LIN {X -0.058,Y -138.324,Z 1253.054,A 0.000,B 0.000,C 90.000,E1 189.670} C_DIS
LIN {X -0.054,Y -139.455,Z 1253.007,A 0.000,B 0.000,C 90.000,E1 181.260} C_DIS
LIN {X 0.026,Y -141.003,Z 1252.976,A 0.000,B 0.000,C 90.000,E1 175.641} C_DIS
LIN {X -0.024,Y -142.757,Z 1252.955,A 0.000,B 0.000,C 90.000,E1 171.951} C_DIS
LIN {X -0.068,Y -145.160,Z 1252.930,A 0.000,B 0.000,C 90.000,E1 167.353} C_DIS
LIN {X -0.076,Y -147.782,Z 1252.909,A 0.000,B 0.000,C 90.000,E1 163.685} C_DIS
LIN {X 0.003,Y -150.461,Z 1252.889,A 0.000,B 0.000,C 90.000,E1 160.007} C_DIS
LIN {X 0.078,Y -153.912,Z 1252.869,A 0.000,B 0.000,C 90.000,E1 156.357} C_DIS
LIN {X 0.002,Y -157.323,Z 1252.849,A 0.000,B 0.000,C 90.000,E1 152.794} C_DIS
LIN {X 0.086,Y -161.512,Z 1252.829,A 0.000,B 0.000,C 90.000,E1 149.203} C_DIS
LIN {X -0.037,Y -165.711,Z 1252.809,A 0.000,B 0.000,C 90.000,E1 145.722} C_DIS
LIN {X 0.088,Y -170.657,Z 1252.790,A 0.000,B 0.000,C 90.000,E1 142.190} C_DIS
LIN {X 0.001,Y -175.532,Z 1252.771,A 0.000,B 0.000,C 90.000,E1 138.771} C_DIS
LIN {X -0.005,Y -181.152,Z 1252.752,A 0.000,B 0.000,C 90.000,E1 135.364} C_DIS
LIN {X -0.007,Y -186.606,Z 1252.733,A 0.000,B 0.000,C 90.000,E1 132.000} C_DIS
LIN {X 0.063,Y -191.215,Z 1252.719,A 0.000,B 0.000,C 90.000,E1 129.483} C_DIS
LIN {X -0.014,Y -197.028,Z 1252.701,A 0.000,B 0.000,C 90.000,E1 126.217} C_DIS
LIN {X 0.090,Y -200.353,Z 1252.692,A 0.000,B 0.000,C 90.000,E1 124.532} C_DIS
LIN {X 0.088,Y -310.121,Z 1252.692,A 0.000,B 0.000,C 90.000,E1 124.532} C_DIS
LIN {X -0.070,Y -311.835,Z 1252.692,A 0.000,B 0.000,C 90.000,E1 124.532} C_DIS
LIN {X 0.041,Y -316.000,Z 1252.691,A 0.000,B 0.000,C 90.000,E1 124.326} C_DIS
LIN {X 0.153,Y -318.367,Z 1252.690,A 0.000,B 0.000,C 90.000,E1 124.119} C_DIS
LIN {X -0.062,Y -321.599,Z 1252.688,A 0.000,B 0.000,C 90.000,E1 123.785} C_DIS
LIN {X 0.072,Y -323.525,Z 1252.686,A 0.000,B 0.000,C 90.000,E1 123.452} C_DIS
LIN {X -0.064,Y -325.025,Z 1252.684,A 0.000,B 0.000,C 90.000,E1 123.166} C_DIS
LIN {X -0.150,Y -339.403,Z 1252.663,A 0.000,B 0.000,C 90.000,E1 119.411} C_DIS
LIN {X 0.030,Y -351.700,Z 1252.648,A 0.000,B 0.000,C 90.000,E1 116.616} C_DIS
LIN {X 0.098,Y -365.488,Z 1252.633,A 0.000,B 0.000,C 90.000,E1 113.898} C_DIS
LIN {X 0.158,Y -379.088,Z 1252.620,A 0.000,B 0.000,C 90.000,E1 111.535} C_DIS
LIN {X -0.083,Y -394.054,Z 1252.607,A 0.000,B 0.000,C 90.000,E1 109.268} C_DIS
LIN {X 0.163,Y -410.491,Z 1252.594,A 0.000,B 0.000,C 90.000,E1 106.985} C_DIS
LIN {X -0.097,Y -428.516,Z 1252.582,A 0.000,B 0.000,C 90.000,E1 104.828} C_DIS
LIN {X -0.031,Y -448.086,Z 1252.571,A 0.000,B 0.000,C 90.000,E1 102.703} C_DIS
LIN {X 0.153,Y -468.363,Z 1252.560,A 0.000,B 0.000,C 90.000,E1 100.725} C_DIS
LIN {X 0.224,Y -473.517,Z 1252.557,A 0.000,B 0.000,C 90.000,E1 100.254} C_DIS
LIN {X -0.170,Y -475.724,Z 1252.556,A 0.000,B 0.000,C 90.000,E1 100.074} C_DIS
LIN {X -0.179,Y -477.397,Z 1252.555,A 0.000,B 0.000,C 90.000,E1 99.849} C_DIS
LIN {X 0.161,Y -478.807,Z 1252.553,A 0.000,B 0.000,C 90.000,E1 99.557} C_DIS
LIN {X 0.031,Y -479.855,Z 1252.552,A 0.000,B 0.000,C 90.000,E1 99.321} C_DIS
LIN {X 0.182,Y -481.069,Z 1252.549,A 0.000,B 0.000,C 90.000,E1 98.803} C_DIS
LIN {X -0.135,Y -481.271,Z 1252.546,A 0.000,B 0.000,C 90.000,E1 98.341} C_DIS
LIN {X 0.100,Y -480.495,Z 1252.543,A 0.000,B 0.000,C 90.000,E1 97.814} C_DIS
LIN {X -0.207,Y -478.616,Z 1252.541,A 0.000,B 0.000,C 90.000,E1 97.352} C_DIS
LIN {X 0.083,Y -477.147,Z 1252.539,A 0.000,B 0.000,C 90.000,E1 97.068} C_DIS
LIN {X 0.209,Y -455.290,Z 1252.522,A 0.000,B 0.000,C 90.000,E1 94.012} C_DIS
LIN {X -0.077,Y -434.881,Z 1252.505,A 0.000,B 0.000,C 90.000,E1 90.917} C_DIS
LIN {X -0.165,Y -416.705,Z 1252.487,A 0.000,B 0.000,C 90.000,E1 87.707} C_DIS
LIN {X 0.075,Y -406.737,Z 1252.476,A 0.000,B 0.000,C 90.000,E1 85.755} C_DIS
LIN {X 0.052,Y -398.078,Z 1252.467,A 0.000,B 0.000,C 90.000,E1 84.090} C_DIS
LIN {X -0.043,Y -387.828,Z 1252.456,A 0.000,B 0.000,C 90.000,E1 82.129} C_DIS
LIN {X 0.121,Y -378.888,Z 1252.447,A 0.000,B 0.000,C 90.000,E1 80.387} C_DIS
LIN {X 0.190,Y -369.652,Z 1252.437,A 0.000,B 0.000,C 90.000,E1 78.634} C_DIS
LIN {X 0.091,Y -360.056,Z 1252.427,A 0.000,B 0.000,C 90.000,E1 76.881} C_DIS
LIN {X -0.076,Y -348.672,Z 1252.416,A 0.000,B 0.000,C 90.000,E1 74.810} C_DIS
LIN {X -0.061,Y -337.274,Z 1252.404,A 0.000,B 0.000,C 90.000,E1 72.670} C_DIS
LIN {X -0.163,Y -323.043,Z 1252.388,A 0.000,B 0.000,C 90.000,E1 69.880} C_DIS
LIN {X 0.099,Y -306.698,Z 1252.368,A 0.000,B 0.000,C 90.000,E1 66.305} C_DIS
LIN {X 0.157,Y -293.245,Z 1252.350,A 0.000,B 0.000,C 90.000,E1 62.999} C_DIS
LIN {X -0.037,Y -281.119,Z 1252.331,A 0.000,B 0.000,C 90.000,E1 59.665} C_DIS
LIN {X 0.048,Y -271.095,Z 1252.314,A 0.000,B 0.000,C 90.000,E1 56.548} C_DIS
LIN {X 0.018,Y -260.896,Z 1252.295,A 0.000,B 0.000,C 90.000,E1 53.050} C_DIS
LIN {X 0.087,Y -251.610,Z 1252.275,A 0.000,B 0.000,C 90.000,E1 49.461} C_DIS
LIN {X 0.138,Y -242.914,Z 1252.255,A 0.000,B 0.000,C 90.000,E1 45.810} C_DIS
LIN {X -0.030,Y -236.363,Z 1252.238,A 0.000,B 0.000,C 90.000,E1 42.894} C_DIS
LIN {X 0.080,Y -228.433,Z 1252.217,A 0.000,B 0.000,C 90.000,E1 39.116} C_DIS
LIN {X 0.051,Y -221.113,Z 1252.196,A 0.000,B 0.000,C 90.000,E1 35.311} C_DIS
LIN {X -0.037,Y -214.422,Z 1252.175,A 0.000,B 0.000,C 90.000,E1 31.465} C_DIS
LIN {X 0.068,Y -208.556,Z 1252.153,A 0.000,B 0.000,C 90.000,E1 27.513} C_DIS
LIN {X -0.025,Y -203.615,Z 1252.131,A 0.000,B 0.000,C 90.000,E1 23.567} C_DIS
LIN {X -0.104,Y -199.415,Z 1252.109,A 0.000,B 0.000,C 90.000,E1 19.577} C_DIS
LIN {X 0.077,Y -195.382,Z 1252.082,A 0.000,B 0.000,C 90.000,E1 14.662} C_DIS
LIN {X -0.039,Y -192.250,Z 1252.050,A 0.000,B 0.000,C 90.000,E1 8.973} C_DIS
LIN {X -0.086,Y -193.147,Z 1251.965,A 0.000,B 0.000,C 90.000,E1 353.799} C_DIS
LIN {X -0.012,Y -196.611,Z 1251.934,A 0.000,B 0.000,C 90.000,E1 348.049} C_DIS
LIN {X -0.074,Y -200.794,Z 1251.906,A 0.000,B 0.000,C 90.000,E1 343.196} C_DIS
LIN {X -0.013,Y -205.052,Z 1251.884,A 0.000,B 0.000,C 90.000,E1 339.156} C_DIS
LIN {X -0.035,Y -210.056,Z 1251.862,A 0.000,B 0.000,C 90.000,E1 335.177} C_DIS
LIN {X -0.114,Y -215.658,Z 1251.840,A 0.000,B 0.000,C 90.000,E1 331.257} C_DIS
LIN {X 0.028,Y -222.004,Z 1251.818,A 0.000,B 0.000,C 90.000,E1 327.327} C_DIS
LIN {X -0.011,Y -228.987,Z 1251.797,A 0.000,B 0.000,C 90.000,E1 323.497} C_DIS
LIN {X 0.032,Y -236.807,Z 1251.776,A 0.000,B 0.000,C 90.000,E1 319.703} C_DIS
LIN {X 0.071,Y -245.561,Z 1251.755,A 0.000,B 0.000,C 90.000,E1 315.972} C_DIS
LIN {X 0.038,Y -254.501,Z 1251.737,A 0.000,B 0.000,C 90.000,E1 312.690} C_DIS
LIN {X 0.007,Y -261.337,Z 1251.725,A 0.000,B 0.000,C 90.000,E1 310.539} C_DIS
LIN {X 0.137,Y -269.058,Z 1251.713,A 0.000,B 0.000,C 90.000,E1 308.382} C_DIS
LIN {X -0.011,Y -276.269,Z 1251.704,A 0.000,B 0.000,C 90.000,E1 306.664} C_DIS
LIN {X 0.035,Y -287.524,Z 1251.690,A 0.000,B 0.000,C 90.000,E1 304.246} C_DIS
LIN {X 0.086,Y -298.162,Z 1251.679,A 0.000,B 0.000,C 90.000,E1 302.212} C_DIS
LIN {X -0.104,Y -308.042,Z 1251.670,A 0.000,B 0.000,C 90.000,E1 300.590} C_DIS
LIN {X -0.090,Y -316.893,Z 1251.663,A 0.000,B 0.000,C 90.000,E1 299.283} C_DIS
LIN {X 0.040,Y -333.695,Z 1251.650,A 0.000,B 0.000,C 90.000,E1 297.052} C_DIS
LIN {X 0.051,Y -354.472,Z 1251.637,A 0.000,B 0.000,C 90.000,E1 294.591} C_DIS
LIN {X 0.129,Y -370.142,Z 1251.627,A 0.000,B 0.000,C 90.000,E1 292.823} C_DIS
LIN {X 0.044,Y -382.927,Z 1251.619,A 0.000,B 0.000,C 90.000,E1 291.408} C_DIS
LIN {X -0.151,Y -400.960,Z 1251.608,A 0.000,B 0.000,C 90.000,E1 289.450} C_DIS
LIN {X 0.050,Y -416.174,Z 1251.599,A 0.000,B 0.000,C 90.000,E1 287.819} C_DIS
LIN {X 0.207,Y -425.892,Z 1251.593,A 0.000,B 0.000,C 90.000,E1 286.732} C_DIS
LIN {X -0.128,Y -432.798,Z 1251.589,A 0.000,B 0.000,C 90.000,E1 285.969} C_DIS
LIN {X 0.122,Y -439.139,Z 1251.584,A 0.000,B 0.000,C 90.000,E1 285.134} C_DIS
LIN {X -0.002,Y -444.874,Z 1251.580,A 0.000,B 0.000,C 90.000,E1 284.356} C_DIS
LIN {X -0.185,Y -449.960,Z 1251.575,A 0.000,B 0.000,C 90.000,E1 283.592} C_DIS
LIN {X 0.114,Y -454.343,Z 1251.571,A 0.000,B 0.000,C 90.000,E1 282.771} C_DIS
LIN {X 0.017,Y -458.046,Z 1251.567,A 0.000,B 0.000,C 90.000,E1 282.007} C_DIS
LIN {X -0.055,Y -461.090,Z 1251.562,A 0.000,B 0.000,C 90.000,E1 281.243} C_DIS
LIN {X 0.056,Y -462.821,Z 1251.560,A 0.000,B 0.000,C 90.000,E1 280.715} C_DIS
LIN {X 0.095,Y -464.245,Z 1251.557,A 0.000,B 0.000,C 90.000,E1 280.197} C_DIS
LIN {X 0.228,Y -465.421,Z 1251.554,A 0.000,B 0.000,C 90.000,E1 279.670} C_DIS
LIN {X -0.170,Y -466.301,Z 1251.551,A 0.000,B 0.000,C 90.000,E1 279.208} C_DIS
LIN {X -0.027,Y -466.922,Z 1251.548,A 0.000,B 0.000,C 90.000,E1 278.681} C_DIS
LIN {X 0.050,Y -467.186,Z 1251.545,A 0.000,B 0.000,C 90.000,E1 278.163} C_DIS
LIN {X 0.133,Y -467.079,Z 1251.543,A 0.000,B 0.000,C 90.000,E1 277.644} C_DIS
LIN {X 0.218,Y -466.525,Z 1251.540,A 0.000,B 0.000,C 90.000,E1 277.125} C_DIS
LIN {X -0.159,Y -465.542,Z 1251.537,A 0.000,B 0.000,C 90.000,E1 276.663} C_DIS
LIN {X -0.076,Y -464.136,Z 1251.534,A 0.000,B 0.000,C 90.000,E1 276.144} C_DIS
LIN {X -0.174,Y -461.221,Z 1251.530,A 0.000,B 0.000,C 90.000,E1 275.391} C_DIS
LIN {X -0.156,Y -458.859,Z 1251.527,A 0.000,B 0.000,C 90.000,E1 274.878} C_DIS
LIN {X -0.114,Y -455.967,Z 1251.524,A 0.000,B 0.000,C 90.000,E1 274.359} C_DIS
LIN {X -0.088,Y -452.395,Z 1251.521,A 0.000,B 0.000,C 90.000,E1 273.841} C_DIS
LIN {X -0.110,Y -447.800,Z 1251.518,A 0.000,B 0.000,C 90.000,E1 273.326} C_DIS
LIN {X 0.121,Y -445.050,Z 1251.517,A 0.000,B 0.000,C 90.000,E1 273.037} C_DIS
LIN {X -0.100,Y -438.896,Z 1251.514,A 0.000,B 0.000,C 90.000,E1 272.579} C_DIS
LIN {X -0.209,Y -432.234,Z 1251.512,A 0.000,B 0.000,C 90.000,E1 272.178} C_DIS
LIN {X -0.199,Y -425.256,Z 1251.510,A 0.000,B 0.000,C 90.000,E1 271.833} C_DIS
LIN {X -0.191,Y -418.174,Z 1251.508,A 0.000,B 0.000,C 90.000,E1 271.547} C_DIS
LIN {X -0.160,Y -407.620,Z 1251.507,A 0.000,B 0.000,C 90.000,E1 271.203} C_DIS
LIN {X 0.154,Y -400.372,Z 1251.505,A 0.000,B 0.000,C 90.000,E1 270.974} C_DIS
LIN {X -0.113,Y -393.101,Z 1251.505,A 0.000,B 0.000,C 90.000,E1 270.859} C_DIS
LIN {X -0.171,Y -384.846,Z 1251.504,A 0.000,B 0.000,C 90.000,E1 270.745} C_DIS
LIN {X 0.169,Y -372.232,Z 1251.503,A 0.000,B 0.000,C 90.000,E1 270.573} C_DIS
LIN {X -0.023,Y -363.644,Z 1251.503,A 0.000,B 0.000,C 90.000,E1 270.573} C_DIS
LIN {X -0.036,Y -181.556,Z 1251.503,A 0.000,B 0.000,C 90.000,E1 270.573} C_DIS
LIN {X -0.072,Y -181.282,Z 1251.494,A 0.000,B 0.000,C 90.000,E1 268.854} C_DIS
LIN {X -0.023,Y -180.907,Z 1251.475,A 0.000,B 0.000,C 90.000,E1 265.469} C_DIS
LIN {X 0.034,Y -180.733,Z 1251.470,A 0.000,B 0.000,C 90.000,E1 264.609} C_DIS
LIN {X -0.044,Y -178.822,Z 1251.442,A 0.000,B 0.000,C 90.000,E1 259.567} C_DIS
LIN {X 0.037,Y -175.868,Z 1251.414,A 0.000,B 0.000,C 90.000,E1 254.448} C_DIS
LIN {X 0.032,Y -173.837,Z 1251.399,A 0.000,B 0.000,C 90.000,E1 251.891} C_DIS
LIN {X 0.021,Y -171.505,Z 1251.380,A 0.000,B 0.000,C 90.000,E1 248.465} C_DIS
LIN {X 0.007,Y -167.732,Z 1251.356,A 0.000,B 0.000,C 90.000,E1 244.152} C_DIS
LIN {X 0.024,Y -166.429,Z 1251.347,A 0.000,B 0.000,C 90.000,E1 242.410} C_DIS
LIN {X 0.021,Y -163.149,Z 1251.327,A 0.000,B 0.000,C 90.000,E1 238.918} C_DIS
LIN {X -0.013,Y -161.105,Z 1251.313,A 0.000,B 0.000,C 90.000,E1 236.294} C_DIS
LIN {X -0.030,Y -157.831,Z 1251.293,A 0.000,B 0.000,C 90.000,E1 232.763} C_DIS
LIN {X 0.034,Y -155.865,Z 1251.278,A 0.000,B 0.000,C 90.000,E1 230.070} C_DIS
LIN {X 0.089,Y -152.115,Z 1251.253,A 0.000,B 0.000,C 90.000,E1 225.567} C_DIS
LIN {X -0.004,Y -150.365,Z 1251.238,A 0.000,B 0.000,C 90.000,E1 222.894} C_DIS
LIN {X 0.035,Y -147.100,Z 1251.213,A 0.000,B 0.000,C 90.000,E1 218.338} C_DIS
LIN {X 0.029,Y -145.669,Z 1251.198,A 0.000,B 0.000,C 90.000,E1 215.598} C_DIS
LIN {X 0.032,Y -143.051,Z 1251.172,A 0.000,B 0.000,C 90.000,E1 211.003} C_DIS
LIN {X -0.032,Y -141.674,Z 1251.152,A 0.000,B 0.000,C 90.000,E1 207.334} C_DIS
LIN {X 0.077,Y -139.454,Z 1251.116,A 0.000,B 0.000,C 90.000,E1 200.791} C_DIS
LIN {X -0.003,Y -139.188,Z 1251.105,A 0.000,B 0.000,C 90.000,E1 198.960} C_DIS
LIN {X 0.020,Y -138.323,Z 1251.053,A 0.000,B 0.000,C 90.000,E1 189.613} C_DIS
LIN {X 0.028,Y -139.458,Z 1251.007,A 0.000,B 0.000,C 90.000,E1 181.203} C_DIS
LIN {X -0.032,Y -141.012,Z 1250.976,A 0.000,B 0.000,C 90.000,E1 175.641} C_DIS
LIN {X 0.059,Y -142.766,Z 1250.955,A 0.000,B 0.000,C 90.000,E1 171.894} C_DIS
LIN {X 0.014,Y -145.175,Z 1250.929,A 0.000,B 0.000,C 90.000,E1 167.297} C_DIS
LIN {X 0.047,Y -147.797,Z 1250.909,A 0.000,B 0.000,C 90.000,E1 163.614} C_DIS
LIN {X -0.057,Y -150.481,Z 1250.889,A 0.000,B 0.000,C 90.000,E1 160.007} C_DIS
LIN {X 0.016,Y -153.935,Z 1250.869,A 0.000,B 0.000,C 90.000,E1 156.357} C_DIS
LIN {X 0.079,Y -157.346,Z 1250.849,A 0.000,B 0.000,C 90.000,E1 152.743} C_DIS
LIN {X 0.023,Y -161.541,Z 1250.829,A 0.000,B 0.000,C 90.000,E1 149.203} C_DIS
LIN {X 0.036,Y -165.739,Z 1250.809,A 0.000,B 0.000,C 90.000,E1 145.674} C_DIS
LIN {X 0.023,Y -170.692,Z 1250.790,A 0.000,B 0.000,C 90.000,E1 142.190} C_DIS
LIN {X -0.065,Y -175.565,Z 1250.771,A 0.000,B 0.000,C 90.000,E1 138.771} C_DIS
LIN {X 0.054,Y -181.184,Z 1250.752,A 0.000,B 0.000,C 90.000,E1 135.324} C_DIS
LIN {X -0.076,Y -186.643,Z 1250.733,A 0.000,B 0.000,C 90.000,E1 132.000} C_DIS
LIN {X -0.008,Y -191.249,Z 1250.719,A 0.000,B 0.000,C 90.000,E1 129.483} C_DIS
LIN {X 0.073,Y -197.068,Z 1250.701,A 0.000,B 0.000,C 90.000,E1 126.171} C_DIS
LIN {X 0.019,Y -200.395,Z 1250.692,A 0.000,B 0.000,C 90.000,E1 124.532} C_DIS
LIN {X -0.024,Y -309.372,Z 1250.692,A 0.000,B 0.000,C 90.000,E1 124.532} C_DIS
LIN {X 0.075,Y -311.716,Z 1250.692,A 0.000,B 0.000,C 90.000,E1 124.485} C_DIS
LIN {X -0.072,Y -315.998,Z 1250.691,A 0.000,B 0.000,C 90.000,E1 124.326} C_DIS
LIN {X 0.040,Y -318.385,Z 1250.690,A 0.000,B 0.000,C 90.000,E1 124.119} C_DIS
LIN {X -0.178,Y -321.634,Z 1250.688,A 0.000,B 0.000,C 90.000,E1 123.785} C_DIS
LIN {X -0.037,Y -323.561,Z 1250.686,A 0.000,B 0.000,C 90.000,E1 123.452} C_DIS
LIN {X -0.168,Y -325.062,Z 1250.684,A 0.000,B 0.000,C 90.000,E1 123.166} C_DIS
LIN {X 0.039,Y -339.456,Z 1250.663,A 0.000,B 0.000,C 90.000,E1 119.361} C_DIS
LIN {X -0.079,Y -351.762,Z 1250.648,A 0.000,B 0.000,C 90.000,E1 116.616} C_DIS
LIN {X -0.013,Y -365.559,Z 1250.633,A 0.000,B 0.000,C 90.000,E1 113.898} C_DIS
LIN {X 0.045,Y -379.169,Z 1250.620,A 0.000,B 0.000,C 90.000,E1 111.535} C_DIS
LIN {X -0.199,Y -394.145,Z 1250.607,A 0.000,B 0.000,C 90.000,E1 109.268} C_DIS
LIN {X 0.044,Y -410.593,Z 1250.594,A 0.000,B 0.000,C 90.000,E1 106.985} C_DIS
LIN {X 0.196,Y -428.629,Z 1250.582,A 0.000,B 0.000,C 90.000,E1 104.773} C_DIS
LIN {X -0.150,Y -448.207,Z 1250.570,A 0.000,B 0.000,C 90.000,E1 102.703} C_DIS
LIN {X 0.125,Y -468.490,Z 1250.560,A 0.000,B 0.000,C 90.000,E1 100.715} C_DIS
LIN {X 0.109,Y -473.641,Z 1250.557,A 0.000,B 0.000,C 90.000,E1 100.254} C_DIS
LIN {X 0.155,Y -475.811,Z 1250.556,A 0.000,B 0.000,C 90.000,E1 100.018} C_DIS
LIN {X 0.120,Y -477.454,Z 1250.554,A 0.000,B 0.000,C 90.000,E1 99.792} C_DIS
LIN {X -0.010,Y -478.818,Z 1250.553,A 0.000,B 0.000,C 90.000,E1 99.557} C_DIS
LIN {X -0.141,Y -479.829,Z 1250.552,A 0.000,B 0.000,C 90.000,E1 99.321} C_DIS
LIN {X 0.010,Y -480.981,Z 1250.549,A 0.000,B 0.000,C 90.000,E1 98.803} C_DIS
LIN {X 0.239,Y -481.128,Z 1250.546,A 0.000,B 0.000,C 90.000,E1 98.276} C_DIS
LIN {X -0.072,Y -480.294,Z 1250.543,A 0.000,B 0.000,C 90.000,E1 97.814} C_DIS
LIN {X 0.095,Y -478.343,Z 1250.541,A 0.000,B 0.000,C 90.000,E1 97.296} C_DIS
LIN {X -0.090,Y -476.826,Z 1250.539,A 0.000,B 0.000,C 90.000,E1 97.068} C_DIS
LIN {X -0.008,Y -458.494,Z 1250.525,A 0.000,B 0.000,C 90.000,E1 94.531} C_DIS
LIN {X 0.108,Y -439.450,Z 1250.509,A 0.000,B 0.000,C 90.000,E1 91.661} C_DIS
LIN {X -0.094,Y -423.737,Z 1250.495,A 0.000,B 0.000,C 90.000,E1 89.026} C_DIS
LIN {X 0.125,Y -409.273,Z 1250.479,A 0.000,B 0.000,C 90.000,E1 86.274} C_DIS
LIN {X 0.146,Y -400.680,Z 1250.470,A 0.000,B 0.000,C 90.000,E1 84.609} C_DIS
LIN {X 0.102,Y -390.447,Z 1250.459,A 0.000,B 0.000,C 90.000,E1 82.648} C_DIS
LIN {X -0.124,Y -381.591,Z 1250.450,A 0.000,B 0.000,C 90.000,E1 80.971} C_DIS
LIN {X -0.006,Y -372.448,Z 1250.440,A 0.000,B 0.000,C 90.000,E1 79.218} C_DIS
LIN {X -0.026,Y -364.591,Z 1250.432,A 0.000,B 0.000,C 90.000,E1 77.757} C_DIS
LIN {X -0.131,Y -354.893,Z 1250.422,A 0.000,B 0.000,C 90.000,E1 75.992} C_DIS
LIN {X -0.069,Y -343.475,Z 1250.410,A 0.000,B 0.000,C 90.000,E1 73.866} C_DIS
LIN {X -0.089,Y -330.597,Z 1250.397,A 0.000,B 0.000,C 90.000,E1 71.402} C_DIS
LIN {X 0.095,Y -318.159,Z 1250.383,A 0.000,B 0.000,C 90.000,E1 68.847} C_DIS
LIN {X 0.021,Y -302.275,Z 1250.363,A 0.000,B 0.000,C 90.000,E1 65.305} C_DIS
LIN {X 0.061,Y -288.037,Z 1250.343,A 0.000,B 0.000,C 90.000,E1 61.641} C_DIS
LIN {X -0.004,Y -276.307,Z 1250.324,A 0.000,B 0.000,C 90.000,E1 58.250} C_DIS
LIN {X 0.108,Y -266.620,Z 1250.306,A 0.000,B 0.000,C 90.000,E1 55.102} C_DIS
LIN {X -0.121,Y -256.771,Z 1250.287,A 0.000,B 0.000,C 90.000,E1 51.618} C_DIS
LIN {X 0.105,Y -249.482,Z 1250.271,A 0.000,B 0.000,C 90.000,E1 48.690} C_DIS
LIN {X -0.085,Y -240.902,Z 1250.250,A 0.000,B 0.000,C 90.000,E1 45.081} C_DIS
LIN {X 0.049,Y -234.325,Z 1250.234,A 0.000,B 0.000,C 90.000,E1 42.081} C_DIS
LIN {X 0.053,Y -228.007,Z 1250.217,A 0.000,B 0.000,C 90.000,E1 39.072} C_DIS
LIN {X 0.021,Y -220.660,Z 1250.196,A 0.000,B 0.000,C 90.000,E1 35.264} C_DIS
LIN {X 0.041,Y -213.939,Z 1250.174,A 0.000,B 0.000,C 90.000,E1 31.386} C_DIS
LIN {X 0.026,Y -208.073,Z 1250.153,A 0.000,B 0.000,C 90.000,E1 27.462} C_DIS
LIN {X -0.073,Y -203.138,Z 1250.130,A 0.000,B 0.000,C 90.000,E1 23.515} C_DIS
LIN {X 0.093,Y -198.951,Z 1250.108,A 0.000,B 0.000,C 90.000,E1 19.450} C_DIS
LIN {X 0.057,Y -194.943,Z 1250.081,A 0.000,B 0.000,C 90.000,E1 14.592} C_DIS
LIN {X 0.069,Y -191.876,Z 1250.049,A 0.000,B 0.000,C 90.000,E1 8.859} C_DIS
LIN {X 0.094,Y -192.895,Z 1249.965,A 0.000,B 0.000,C 90.000,E1 353.742} C_DIS
LIN {X -0.034,Y -196.381,Z 1249.934,A 0.000,B 0.000,C 90.000,E1 348.049} C_DIS
LIN {X 0.086,Y -200.590,Z 1249.906,A 0.000,B 0.000,C 90.000,E1 343.142} C_DIS
LIN {X 0.022,Y -204.905,Z 1249.884,A 0.000,B 0.000,C 90.000,E1 339.135} C_DIS
LIN {X 0.010,Y -209.920,Z 1249.862,A 0.000,B 0.000,C 90.000,E1 335.153} C_DIS
LIN {X 0.131,Y -215.545,Z 1249.840,A 0.000,B 0.000,C 90.000,E1 331.179} C_DIS
LIN {X -0.025,Y -221.928,Z 1249.818,A 0.000,B 0.000,C 90.000,E1 327.327} C_DIS
LIN {X -0.068,Y -228.914,Z 1249.797,A 0.000,B 0.000,C 90.000,E1 323.497} C_DIS
LIN {X -0.030,Y -236.736,Z 1249.776,A 0.000,B 0.000,C 90.000,E1 319.703} C_DIS
LIN {X 0.005,Y -245.497,Z 1249.755,A 0.000,B 0.000,C 90.000,E1 315.972} C_DIS
LIN {X -0.032,Y -254.428,Z 1249.737,A 0.000,B 0.000,C 90.000,E1 312.690} C_DIS
LIN {X -0.067,Y -261.268,Z 1249.725,A 0.000,B 0.000,C 90.000,E1 310.539} C_DIS
LIN {X 0.060,Y -269.017,Z 1249.713,A 0.000,B 0.000,C 90.000,E1 308.382} C_DIS
LIN {X -0.090,Y -276.247,Z 1249.704,A 0.000,B 0.000,C 90.000,E1 306.664} C_DIS
LIN {X -0.049,Y -287.473,Z 1249.690,A 0.000,B 0.000,C 90.000,E1 304.246} C_DIS
LIN {X -0.002,Y -298.107,Z 1249.679,A 0.000,B 0.000,C 90.000,E1 302.212} C_DIS
LIN {X 0.070,Y -307.988,Z 1249.670,A 0.000,B 0.000,C 90.000,E1 300.541} C_DIS
LIN {X -0.174,Y -316.783,Z 1249.662,A 0.000,B 0.000,C 90.000,E1 299.283} C_DIS
LIN {X 0.011,Y -326.243,Z 1249.655,A 0.000,B 0.000,C 90.000,E1 297.975} C_DIS
LIN {X 0.077,Y -349.262,Z 1249.640,A 0.000,B 0.000,C 90.000,E1 295.155} C_DIS
LIN {X -0.076,Y -365.142,Z 1249.630,A 0.000,B 0.000,C 90.000,E1 293.387} C_DIS
LIN {X 0.197,Y -378.202,Z 1249.622,A 0.000,B 0.000,C 90.000,E1 291.897} C_DIS
LIN {X 0.086,Y -391.038,Z 1249.614,A 0.000,B 0.000,C 90.000,E1 290.482} C_DIS
LIN {X 0.002,Y -411.509,Z 1249.602,A 0.000,B 0.000,C 90.000,E1 288.308} C_DIS
LIN {X -0.059,Y -419.120,Z 1249.597,A 0.000,B 0.000,C 90.000,E1 287.511} C_DIS
LIN {X 0.101,Y -426.431,Z 1249.593,A 0.000,B 0.000,C 90.000,E1 286.677} C_DIS
LIN {X -0.127,Y -433.306,Z 1249.588,A 0.000,B 0.000,C 90.000,E1 285.898} C_DIS
LIN {X 0.125,Y -439.607,Z 1249.584,A 0.000,B 0.000,C 90.000,E1 285.064} C_DIS
LIN {X -0.111,Y -445.318,Z 1249.579,A 0.000,B 0.000,C 90.000,E1 284.300} C_DIS
LIN {X 0.149,Y -450.332,Z 1249.575,A 0.000,B 0.000,C 90.000,E1 283.480} C_DIS
LIN {X 0.015,Y -454.677,Z 1249.571,A 0.000,B 0.000,C 90.000,E1 282.715} C_DIS
LIN {X -0.080,Y -458.304,Z 1249.566,A 0.000,B 0.000,C 90.000,E1 281.951} C_DIS
LIN {X -0.149,Y -461.305,Z 1249.562,A 0.000,B 0.000,C 90.000,E1 281.186} C_DIS
LIN {X -0.035,Y -463.003,Z 1249.559,A 0.000,B 0.000,C 90.000,E1 280.658} C_DIS
LIN {X 0.005,Y -464.401,Z 1249.556,A 0.000,B 0.000,C 90.000,E1 280.141} C_DIS
LIN {X 0.139,Y -465.529,Z 1249.553,A 0.000,B 0.000,C 90.000,E1 279.613} C_DIS
LIN {X -0.257,Y -466.390,Z 1249.551,A 0.000,B 0.000,C 90.000,E1 279.151} C_DIS
LIN {X -0.113,Y -467.018,Z 1249.548,A 0.000,B 0.000,C 90.000,E1 278.624} C_DIS
LIN {X -0.035,Y -467.268,Z 1249.545,A 0.000,B 0.000,C 90.000,E1 278.106} C_DIS
LIN {X 0.049,Y -467.126,Z 1249.542,A 0.000,B 0.000,C 90.000,E1 277.587} C_DIS
LIN {X 0.136,Y -466.567,Z 1249.539,A 0.000,B 0.000,C 90.000,E1 277.068} C_DIS
LIN {X -0.241,Y -465.557,Z 1249.536,A 0.000,B 0.000,C 90.000,E1 276.606} C_DIS
LIN {X -0.157,Y -464.106,Z 1249.534,A 0.000,B 0.000,C 90.000,E1 276.087} C_DIS
LIN {X 0.206,Y -461.146,Z 1249.529,A 0.000,B 0.000,C 90.000,E1 275.277} C_DIS
LIN {X 0.037,Y -457.304,Z 1249.525,A 0.000,B 0.000,C 90.000,E1 274.531} C_DIS
LIN {X -0.192,Y -455.789,Z 1249.524,A 0.000,B 0.000,C 90.000,E1 274.302} C_DIS
LIN {X -0.167,Y -452.094,Z 1249.521,A 0.000,B 0.000,C 90.000,E1 273.784} C_DIS
LIN {X -0.189,Y -447.430,Z 1249.518,A 0.000,B 0.000,C 90.000,E1 273.269} C_DIS
LIN {X -0.031,Y -441.682,Z 1249.515,A 0.000,B 0.000,C 90.000,E1 272.751} C_DIS
LIN {X -0.100,Y -438.490,Z 1249.514,A 0.000,B 0.000,C 90.000,E1 272.522} C_DIS
LIN {X -0.199,Y -431.662,Z 1249.512,A 0.000,B 0.000,C 90.000,E1 272.121} C_DIS
LIN {X -0.145,Y -424.631,Z 1249.510,A 0.000,B 0.000,C 90.000,E1 271.776} C_DIS
LIN {X -0.095,Y -417.504,Z 1249.508,A 0.000,B 0.000,C 90.000,E1 271.489} C_DIS
LIN {X 0.005,Y -407.161,Z 1249.506,A 0.000,B 0.000,C 90.000,E1 271.146} C_DIS
LIN {X 0.186,Y -396.224,Z 1249.505,A 0.000,B 0.000,C 90.000,E1 270.859} C_DIS
LIN {X 0.020,Y -388.400,Z 1249.504,A 0.000,B 0.000,C 90.000,E1 270.745} C_DIS
LIN {X 0.052,Y -379.512,Z 1249.504,A 0.000,B 0.000,C 90.000,E1 270.630} C_DIS
LIN {X -0.077,Y -368.342,Z 1249.503,A 0.000,B 0.000,C 90.000,E1 270.573} C_DIS
LIN {X -0.146,Y -363.509,Z 1249.503,A 0.000,B 0.000,C 90.000,E1 270.573} C_DIS
LIN {X 0.089,Y -181.558,Z 1249.503,A 0.000,B 0.000,C 90.000,E1 270.516} C_DIS
LIN {X 0.066,Y -181.279,Z 1249.493,A 0.000,B 0.000,C 90.000,E1 268.797} C_DIS
LIN {X -0.066,Y -180.907,Z 1249.475,A 0.000,B 0.000,C 90.000,E1 265.469} C_DIS
LIN {X -0.010,Y -180.726,Z 1249.470,A 0.000,B 0.000,C 90.000,E1 264.609} C_DIS
LIN {X 0.087,Y -178.815,Z 1249.442,A 0.000,B 0.000,C 90.000,E1 259.511} C_DIS
LIN {X -0.006,Y -175.860,Z 1249.414,A 0.000,B 0.000,C 90.000,E1 254.448} C_DIS
LIN {X 0.043,Y -173.827,Z 1249.399,A 0.000,B 0.000,C 90.000,E1 251.873} C_DIS
LIN {X -0.022,Y -171.493,Z 1249.380,A 0.000,B 0.000,C 90.000,E1 248.465} C_DIS
LIN {X -0.034,Y -167.721,Z 1249.356,A 0.000,B 0.000,C 90.000,E1 244.152} C_DIS
LIN {X -0.018,Y -166.415,Z 1249.347,A 0.000,B 0.000,C 90.000,E1 242.410} C_DIS
LIN {X -0.019,Y -163.137,Z 1249.327,A 0.000,B 0.000,C 90.000,E1 238.918} C_DIS
LIN {X -0.054,Y -161.091,Z 1249.313,A 0.000,B 0.000,C 90.000,E1 236.294} C_DIS
LIN {X -0.070,Y -157.820,Z 1249.293,A 0.000,B 0.000,C 90.000,E1 232.763} C_DIS
LIN {X -0.007,Y -155.854,Z 1249.278,A 0.000,B 0.000,C 90.000,E1 230.070} C_DIS
LIN {X 0.050,Y -152.104,Z 1249.253,A 0.000,B 0.000,C 90.000,E1 225.567} C_DIS
LIN {X 0.068,Y -150.355,Z 1249.238,A 0.000,B 0.000,C 90.000,E1 222.852} C_DIS
LIN {X -0.003,Y -147.091,Z 1249.213,A 0.000,B 0.000,C 90.000,E1 218.338} C_DIS
LIN {X -0.009,Y -145.662,Z 1249.198,A 0.000,B 0.000,C 90.000,E1 215.598} C_DIS
LIN {X -0.005,Y -143.044,Z 1249.172,A 0.000,B 0.000,C 90.000,E1 211.003} C_DIS
LIN {X -0.005,Y -141.668,Z 1249.152,A 0.000,B 0.000,C 90.000,E1 207.308} C_DIS
LIN {X 0.040,Y -139.451,Z 1249.116,A 0.000,B 0.000,C 90.000,E1 200.791} C_DIS
LIN {X -0.040,Y -139.185,Z 1249.105,A 0.000,B 0.000,C 90.000,E1 198.960} C_DIS
LIN {X -0.017,Y -138.321,Z 1249.053,A 0.000,B 0.000,C 90.000,E1 189.613} C_DIS
LIN {X -0.009,Y -139.462,Z 1249.007,A 0.000,B 0.000,C 90.000,E1 181.203} C_DIS
LIN {X -0.070,Y -141.019,Z 1248.976,A 0.000,B 0.000,C 90.000,E1 175.641} C_DIS
LIN {X 0.026,Y -142.382,Z 1248.960,A 0.000,B 0.000,C 90.000,E1 172.818} C_DIS
LIN {X -0.053,Y -144.613,Z 1248.934,A 0.000,B 0.000,C 90.000,E1 168.229} C_DIS
LIN {X 0.009,Y -147.807,Z 1248.909,A 0.000,B 0.000,C 90.000,E1 163.614} C_DIS
LIN {X 0.045,Y -150.494,Z 1248.889,A 0.000,B 0.000,C 90.000,E1 159.953} C_DIS
LIN {X -0.024,Y -153.950,Z 1248.869,A 0.000,B 0.000,C 90.000,E1 156.357} C_DIS
LIN {X 0.039,Y -157.362,Z 1248.849,A 0.000,B 0.000,C 90.000,E1 152.743} C_DIS
LIN {X -0.018,Y -161.560,Z 1248.829,A 0.000,B 0.000,C 90.000,E1 149.203} C_DIS
LIN {X -0.006,Y -165.758,Z 1248.809,A 0.000,B 0.000,C 90.000,E1 145.674} C_DIS
LIN {X -0.020,Y -170.714,Z 1248.790,A 0.000,B 0.000,C 90.000,E1 142.190} C_DIS
LIN {X 0.023,Y -175.587,Z 1248.771,A 0.000,B 0.000,C 90.000,E1 138.728} C_DIS
LIN {X 0.011,Y -181.204,Z 1248.752,A 0.000,B 0.000,C 90.000,E1 135.324} C_DIS
LIN {X 0.004,Y -186.668,Z 1248.733,A 0.000,B 0.000,C 90.000,E1 131.962} C_DIS
LIN {X -0.053,Y -191.270,Z 1248.719,A 0.000,B 0.000,C 90.000,E1 129.483} C_DIS
LIN {X 0.027,Y -197.094,Z 1248.701,A 0.000,B 0.000,C 90.000,E1 126.171} C_DIS
LIN {X 0.069,Y -200.460,Z 1248.692,A 0.000,B 0.000,C 90.000,E1 124.485} C_DIS
LIN {X 0.055,Y -310.542,Z 1248.692,A 0.000,B 0.000,C 90.000,E1 124.485} C_DIS
LIN {X -0.146,Y -315.875,Z 1248.691,A 0.000,B 0.000,C 90.000,E1 124.326} C_DIS
LIN {X -0.034,Y -318.319,Z 1248.690,A 0.000,B 0.000,C 90.000,E1 124.119} C_DIS
LIN {X 0.195,Y -321.613,Z 1248.688,A 0.000,B 0.000,C 90.000,E1 123.706} C_DIS
LIN {X 0.083,Y -323.544,Z 1248.686,A 0.000,B 0.000,C 90.000,E1 123.420} C_DIS
LIN {X -0.208,Y -325.050,Z 1248.684,A 0.000,B 0.000,C 90.000,E1 123.166} C_DIS
LIN {X 0.026,Y -338.181,Z 1248.665,A 0.000,B 0.000,C 90.000,E1 119.667} C_DIS
LIN {X 0.170,Y -350.335,Z 1248.649,A 0.000,B 0.000,C 90.000,E1 116.873} C_DIS
LIN {X -0.123,Y -363.961,Z 1248.634,A 0.000,B 0.000,C 90.000,E1 114.207} C_DIS
LIN {X -0.111,Y -377.411,Z 1248.621,A 0.000,B 0.000,C 90.000,E1 111.844} C_DIS
LIN {X 0.098,Y -392.214,Z 1248.608,A 0.000,B 0.000,C 90.000,E1 109.504} C_DIS
LIN {X -0.091,Y -408.475,Z 1248.596,A 0.000,B 0.000,C 90.000,E1 107.275} C_DIS
LIN {X -0.005,Y -426.310,Z 1248.584,A 0.000,B 0.000,C 90.000,E1 105.064} C_DIS
LIN {X -0.033,Y -445.733,Z 1248.572,A 0.000,B 0.000,C 90.000,E1 102.939} C_DIS
LIN {X 0.080,Y -465.948,Z 1248.561,A 0.000,B 0.000,C 90.000,E1 100.950} C_DIS
LIN {X 0.060,Y -473.671,Z 1248.557,A 0.000,B 0.000,C 90.000,E1 100.254} C_DIS
LIN {X 0.104,Y -475.802,Z 1248.556,A 0.000,B 0.000,C 90.000,E1 100.018} C_DIS
LIN {X 0.065,Y -477.419,Z 1248.554,A 0.000,B 0.000,C 90.000,E1 99.792} C_DIS
LIN {X -0.065,Y -478.760,Z 1248.553,A 0.000,B 0.000,C 90.000,E1 99.557} C_DIS
LIN {X -0.196,Y -479.752,Z 1248.552,A 0.000,B 0.000,C 90.000,E1 99.321} C_DIS
LIN {X -0.046,Y -480.871,Z 1248.549,A 0.000,B 0.000,C 90.000,E1 98.803} C_DIS
LIN {X 0.183,Y -480.989,Z 1248.546,A 0.000,B 0.000,C 90.000,E1 98.276} C_DIS
LIN {X -0.128,Y -480.126,Z 1248.543,A 0.000,B 0.000,C 90.000,E1 97.814} C_DIS
LIN {X 0.038,Y -478.137,Z 1248.541,A 0.000,B 0.000,C 90.000,E1 97.296} C_DIS
LIN {X -0.148,Y -476.595,Z 1248.539,A 0.000,B 0.000,C 90.000,E1 97.068} C_DIS
LIN {X 0.167,Y -456.485,Z 1248.524,A 0.000,B 0.000,C 90.000,E1 94.245} C_DIS
LIN {X -0.051,Y -435.954,Z 1248.506,A 0.000,B 0.000,C 90.000,E1 91.146} C_DIS
LIN {X -0.106,Y -417.583,Z 1248.488,A 0.000,B 0.000,C 90.000,E1 87.936} C_DIS
LIN {X -0.125,Y -404.792,Z 1248.475,A 0.000,B 0.000,C 90.000,E1 85.469} C_DIS
LIN {X -0.113,Y -394.597,Z 1248.464,A 0.000,B 0.000,C 90.000,E1 83.514} C_DIS
LIN {X 0.158,Y -384.336,Z 1248.453,A 0.000,B 0.000,C 90.000,E1 81.489} C_DIS
LIN {X -0.127,Y -376.839,Z 1248.445,A 0.000,B 0.000,C 90.000,E1 80.095} C_DIS
LIN {X -0.088,Y -367.548,Z 1248.435,A 0.000,B 0.000,C 90.000,E1 78.342} C_DIS
LIN {X 0.129,Y -357.965,Z 1248.425,A 0.000,B 0.000,C 90.000,E1 76.533} C_DIS
LIN {X 0.000,Y -346.526,Z 1248.414,A 0.000,B 0.000,C 90.000,E1 74.448} C_DIS
LIN {X -0.040,Y -333.608,Z 1248.400,A 0.000,B 0.000,C 90.000,E1 72.000} C_DIS
LIN {X -0.189,Y -321.047,Z 1248.386,A 0.000,B 0.000,C 90.000,E1 69.518} C_DIS
LIN {X 0.130,Y -304.915,Z 1248.366,A 0.000,B 0.000,C 90.000,E1 65.921} C_DIS
LIN {X 0.128,Y -290.346,Z 1248.346,A 0.000,B 0.000,C 90.000,E1 62.281} C_DIS
LIN {X -0.009,Y -278.376,Z 1248.327,A 0.000,B 0.000,C 90.000,E1 58.918} C_DIS
LIN {X 0.009,Y -268.486,Z 1248.310,A 0.000,B 0.000,C 90.000,E1 55.801} C_DIS
LIN {X 0.046,Y -258.391,Z 1248.290,A 0.000,B 0.000,C 90.000,E1 52.271} C_DIS
LIN {X 0.002,Y -249.189,Z 1248.271,A 0.000,B 0.000,C 90.000,E1 48.690} C_DIS
LIN {X -0.024,Y -240.593,Z 1248.250,A 0.000,B 0.000,C 90.000,E1 45.040} C_DIS
LIN {X -0.065,Y -233.974,Z 1248.234,A 0.000,B 0.000,C 90.000,E1 42.081} C_DIS
LIN {X -0.023,Y -226.085,Z 1248.213,A 0.000,B 0.000,C 90.000,E1 38.302} C_DIS
LIN {X -0.072,Y -218.814,Z 1248.192,A 0.000,B 0.000,C 90.000,E1 34.485} C_DIS
LIN {X -0.045,Y -212.245,Z 1248.170,A 0.000,B 0.000,C 90.000,E1 30.590} C_DIS
LIN {X 0.074,Y -206.579,Z 1248.148,A 0.000,B 0.000,C 90.000,E1 26.616} C_DIS
LIN {X 0.023,Y -201.784,Z 1248.126,A 0.000,B 0.000,C 90.000,E1 22.642} C_DIS
LIN {X -0.033,Y -197.026,Z 1248.099,A 0.000,B 0.000,C 90.000,E1 17.819} C_DIS
LIN {X -0.057,Y -193.505,Z 1248.072,A 0.000,B 0.000,C 90.000,E1 12.939} C_DIS
LIN {X -0.062,Y -190.839,Z 1248.035,A 0.000,B 0.000,C 90.000,E1 6.372} C_DIS
LIN {X -0.067,Y -192.258,Z 1247.970,A 0.000,B 0.000,C 90.000,E1 354.609} C_DIS
LIN {X -0.071,Y -195.559,Z 1247.938,A 0.000,B 0.000,C 90.000,E1 348.870} C_DIS
LIN {X -0.032,Y -199.595,Z 1247.911,A 0.000,B 0.000,C 90.000,E1 343.976} C_DIS
LIN {X -0.003,Y -203.824,Z 1247.889,A 0.000,B 0.000,C 90.000,E1 339.934} C_DIS
LIN {X 0.059,Y -208.733,Z 1247.866,A 0.000,B 0.000,C 90.000,E1 335.921} C_DIS
LIN {X 0.039,Y -214.249,Z 1247.844,A 0.000,B 0.000,C 90.000,E1 331.975} C_DIS
LIN {X 0.028,Y -220.496,Z 1247.823,A 0.000,B 0.000,C 90.000,E1 328.074} C_DIS
LIN {X 0.130,Y -227.375,Z 1247.801,A 0.000,B 0.000,C 90.000,E1 324.196} C_DIS
LIN {X -0.016,Y -234.994,Z 1247.780,A 0.000,B 0.000,C 90.000,E1 320.436} C_DIS
LIN {X -0.020,Y -243.581,Z 1247.759,A 0.000,B 0.000,C 90.000,E1 316.701} C_DIS
LIN {X 0.053,Y -252.276,Z 1247.741,A 0.000,B 0.000,C 90.000,E1 313.380} C_DIS
LIN {X 0.011,Y -259.986,Z 1247.727,A 0.000,B 0.000,C 90.000,E1 310.862} C_DIS
LIN {X -0.089,Y -267.616,Z 1247.715,A 0.000,B 0.000,C 90.000,E1 308.749} C_DIS
LIN {X 0.125,Y -274.703,Z 1247.705,A 0.000,B 0.000,C 90.000,E1 306.950} C_DIS
LIN {X 0.135,Y -285.757,Z 1247.692,A 0.000,B 0.000,C 90.000,E1 304.532} C_DIS
LIN {X -0.092,Y -296.206,Z 1247.681,A 0.000,B 0.000,C 90.000,E1 302.546} C_DIS
LIN {X -0.051,Y -305.815,Z 1247.672,A 0.000,B 0.000,C 90.000,E1 300.875} C_DIS
LIN {X 0.095,Y -314.406,Z 1247.664,A 0.000,B 0.000,C 90.000,E1 299.539} C_DIS
LIN {X -0.066,Y -323.730,Z 1247.657,A 0.000,B 0.000,C 90.000,E1 298.281} C_DIS
LIN {X 0.080,Y -341.339,Z 1247.645,A 0.000,B 0.000,C 90.000,E1 296.052} C_DIS
LIN {X -0.059,Y -359.821,Z 1247.633,A 0.000,B 0.000,C 90.000,E1 293.951} C_DIS
LIN {X 0.053,Y -375.426,Z 1247.623,A 0.000,B 0.000,C 90.000,E1 292.206} C_DIS
LIN {X -0.064,Y -388.339,Z 1247.615,A 0.000,B 0.000,C 90.000,E1 290.791} C_DIS
LIN {X 0.198,Y -408.872,Z 1247.603,A 0.000,B 0.000,C 90.000,E1 288.544} C_DIS
LIN {X -0.091,Y -419.077,Z 1247.597,A 0.000,B 0.000,C 90.000,E1 287.511} C_DIS
LIN {X 0.079,Y -426.407,Z 1247.593,A 0.000,B 0.000,C 90.000,E1 286.677} C_DIS
LIN {X -0.155,Y -433.273,Z 1247.588,A 0.000,B 0.000,C 90.000,E1 285.898} C_DIS
LIN {X 0.096,Y -439.599,Z 1247.584,A 0.000,B 0.000,C 90.000,E1 285.064} C_DIS
LIN {X -0.140,Y -445.298,Z 1247.579,A 0.000,B 0.000,C 90.000,E1 284.300} C_DIS
LIN {X 0.119,Y -450.316,Z 1247.575,A 0.000,B 0.000,C 90.000,E1 283.480} C_DIS
LIN {X -0.017,Y -454.675,Z 1247.571,A 0.000,B 0.000,C 90.000,E1 282.715} C_DIS
LIN {X -0.111,Y -458.305,Z 1247.566,A 0.000,B 0.000,C 90.000,E1 281.951} C_DIS
LIN {X -0.180,Y -461.280,Z 1247.562,A 0.000,B 0.000,C 90.000,E1 281.186} C_DIS
LIN {X -0.067,Y -462.968,Z 1247.559,A 0.000,B 0.000,C 90.000,E1 280.658} C_DIS
LIN {X -0.027,Y -464.396,Z 1247.556,A 0.000,B 0.000,C 90.000,E1 280.141} C_DIS
LIN {X 0.107,Y -465.535,Z 1247.553,A 0.000,B 0.000,C 90.000,E1 279.613} C_DIS
LIN {X 0.172,Y -466.403,Z 1247.551,A 0.000,B 0.000,C 90.000,E1 279.095} C_DIS
LIN {X -0.145,Y -467.026,Z 1247.548,A 0.000,B 0.000,C 90.000,E1 278.624} C_DIS
LIN {X -0.067,Y -467.289,Z 1247.545,A 0.000,B 0.000,C 90.000,E1 278.106} C_DIS
LIN {X 0.017,Y -467.214,Z 1247.542,A 0.000,B 0.000,C 90.000,E1 277.587} C_DIS
LIN {X 0.104,Y -466.666,Z 1247.539,A 0.000,B 0.000,C 90.000,E1 277.068} C_DIS
LIN {X 0.190,Y -465.697,Z 1247.536,A 0.000,B 0.000,C 90.000,E1 276.549} C_DIS
LIN {X -0.187,Y -464.258,Z 1247.534,A 0.000,B 0.000,C 90.000,E1 276.087} C_DIS
LIN {X 0.176,Y -461.344,Z 1247.529,A 0.000,B 0.000,C 90.000,E1 275.277} C_DIS
LIN {X 0.009,Y -457.513,Z 1247.525,A 0.000,B 0.000,C 90.000,E1 274.531} C_DIS
LIN {X 0.041,Y -454.247,Z 1247.522,A 0.000,B 0.000,C 90.000,E1 274.012} C_DIS
LIN {X 0.027,Y -450.139,Z 1247.519,A 0.000,B 0.000,C 90.000,E1 273.498} C_DIS
LIN {X -0.213,Y -447.688,Z 1247.518,A 0.000,B 0.000,C 90.000,E1 273.269} C_DIS
LIN {X -0.056,Y -441.986,Z 1247.515,A 0.000,B 0.000,C 90.000,E1 272.751} C_DIS
LIN {X -0.128,Y -438.778,Z 1247.514,A 0.000,B 0.000,C 90.000,E1 272.522} C_DIS
LIN {X -0.218,Y -432.022,Z 1247.512,A 0.000,B 0.000,C 90.000,E1 272.121} C_DIS
LIN {X -0.162,Y -425.079,Z 1247.510,A 0.000,B 0.000,C 90.000,E1 271.776} C_DIS
LIN {X -0.092,Y -418.140,Z 1247.508,A 0.000,B 0.000,C 90.000,E1 271.489} C_DIS
LIN {X -0.120,Y -411.154,Z 1247.507,A 0.000,B 0.000,C 90.000,E1 271.260} C_DIS
LIN {X -0.098,Y -400.472,Z 1247.505,A 0.000,B 0.000,C 90.000,E1 270.974} C_DIS
LIN {X 0.037,Y -393.009,Z 1247.505,A 0.000,B 0.000,C 90.000,E1 270.802} C_DIS
LIN {X -0.040,Y -384.792,Z 1247.504,A 0.000,B 0.000,C 90.000,E1 270.688} C_DIS
LIN {X 0.049,Y -375.546,Z 1247.503,A 0.000,B 0.000,C 90.000,E1 270.573} C_DIS
LIN {X 0.082,Y -362.162,Z 1247.503,A 0.000,B 0.000,C 90.000,E1 270.516} C_DIS
LIN {X 0.018,Y -181.562,Z 1247.503,A 0.000,B 0.000,C 90.000,E1 270.516} C_DIS
LIN {X -0.006,Y -181.274,Z 1247.493,A 0.000,B 0.000,C 90.000,E1 268.797} C_DIS
LIN {X 0.042,Y -180.906,Z 1247.475,A 0.000,B 0.000,C 90.000,E1 265.412} C_DIS
LIN {X -0.081,Y -180.716,Z 1247.470,A 0.000,B 0.000,C 90.000,E1 264.609} C_DIS
LIN {X 0.016,Y -178.803,Z 1247.442,A 0.000,B 0.000,C 90.000,E1 259.511} C_DIS
LIN {X 0.093,Y -175.848,Z 1247.413,A 0.000,B 0.000,C 90.000,E1 254.393} C_DIS
LIN {X 0.052,Y -172.584,Z 1247.390,A 0.000,B 0.000,C 90.000,E1 250.134} C_DIS
LIN {X 0.068,Y -171.474,Z 1247.380,A 0.000,B 0.000,C 90.000,E1 248.411} C_DIS
LIN {X 0.048,Y -167.704,Z 1247.356,A 0.000,B 0.000,C 90.000,E1 244.101} C_DIS
LIN {X 0.061,Y -166.391,Z 1247.347,A 0.000,B 0.000,C 90.000,E1 242.359} C_DIS
LIN {X 0.052,Y -163.118,Z 1247.327,A 0.000,B 0.000,C 90.000,E1 238.869} C_DIS
LIN {X 0.102,Y -161.067,Z 1247.313,A 0.000,B 0.000,C 90.000,E1 236.215} C_DIS
LIN {X -0.011,Y -157.800,Z 1247.293,A 0.000,B 0.000,C 90.000,E1 232.718} C_DIS
LIN {X -0.072,Y -155.836,Z 1247.278,A 0.000,B 0.000,C 90.000,E1 230.070} C_DIS
LIN {X -0.015,Y -152.086,Z 1247.253,A 0.000,B 0.000,C 90.000,E1 225.567} C_DIS
LIN {X 0.004,Y -150.337,Z 1247.238,A 0.000,B 0.000,C 90.000,E1 222.852} C_DIS
LIN {X 0.024,Y -147.077,Z 1247.213,A 0.000,B 0.000,C 90.000,E1 218.302} C_DIS
LIN {X -0.071,Y -145.650,Z 1247.198,A 0.000,B 0.000,C 90.000,E1 215.598} C_DIS
LIN {X -0.068,Y -143.033,Z 1247.172,A 0.000,B 0.000,C 90.000,E1 211.003} C_DIS
LIN {X 0.059,Y -141.657,Z 1247.152,A 0.000,B 0.000,C 90.000,E1 207.257} C_DIS
LIN {X -0.022,Y -139.447,Z 1247.115,A 0.000,B 0.000,C 90.000,E1 200.791} C_DIS
LIN {X 0.031,Y -139.180,Z 1247.105,A 0.000,B 0.000,C 90.000,E1 198.906} C_DIS
LIN {X 0.059,Y -138.320,Z 1247.053,A 0.000,B 0.000,C 90.000,E1 189.557} C_DIS
LIN {X 0.068,Y -139.465,Z 1247.006,A 0.000,B 0.000,C 90.000,E1 181.146} C_DIS
LIN {X 0.010,Y -141.029,Z 1246.975,A 0.000,B 0.000,C 90.000,E1 175.584} C_DIS
LIN {X -0.036,Y -142.396,Z 1246.960,A 0.000,B 0.000,C 90.000,E1 172.818} C_DIS
LIN {X 0.026,Y -144.628,Z 1246.934,A 0.000,B 0.000,C 90.000,E1 168.173} C_DIS
LIN {X -0.055,Y -147.823,Z 1246.909,A 0.000,B 0.000,C 90.000,E1 163.614} C_DIS
LIN {X 0.031,Y -150.514,Z 1246.889,A 0.000,B 0.000,C 90.000,E1 159.934} C_DIS
LIN {X 0.052,Y -153.976,Z 1246.868,A 0.000,B 0.000,C 90.000,E1 156.305} C_DIS
LIN {X -0.028,Y -157.388,Z 1246.849,A 0.000,B 0.000,C 90.000,E1 152.743} C_DIS
LIN {X -0.086,Y -161.591,Z 1246.829,A 0.000,B 0.000,C 90.000,E1 149.203} C_DIS
LIN {X -0.075,Y -165.789,Z 1246.809,A 0.000,B 0.000,C 90.000,E1 145.674} C_DIS
LIN {X -0.090,Y -170.751,Z 1246.790,A 0.000,B 0.000,C 90.000,E1 142.190} C_DIS
LIN {X 0.068,Y -175.623,Z 1246.771,A 0.000,B 0.000,C 90.000,E1 138.690} C_DIS
LIN {X -0.062,Y -181.238,Z 1246.752,A 0.000,B 0.000,C 90.000,E1 135.324} C_DIS
LIN {X 0.069,Y -186.708,Z 1246.733,A 0.000,B 0.000,C 90.000,E1 131.919} C_DIS
LIN {X 0.020,Y -191.308,Z 1246.719,A 0.000,B 0.000,C 90.000,E1 129.439} C_DIS
LIN {X -0.049,Y -197.137,Z 1246.701,A 0.000,B 0.000,C 90.000,E1 126.171} C_DIS
LIN {X -0.007,Y -200.503,Z 1246.692,A 0.000,B 0.000,C 90.000,E1 124.485} C_DIS
LIN {X -0.064,Y -310.193,Z 1246.692,A 0.000,B 0.000,C 90.000,E1 124.485} C_DIS
LIN {X -0.006,Y -315.878,Z 1246.690,A 0.000,B 0.000,C 90.000,E1 124.278} C_DIS
LIN {X -0.156,Y -318.343,Z 1246.689,A 0.000,B 0.000,C 90.000,E1 124.119} C_DIS
LIN {X 0.072,Y -321.653,Z 1246.687,A 0.000,B 0.000,C 90.000,E1 123.706} C_DIS
LIN {X -0.034,Y -323.584,Z 1246.686,A 0.000,B 0.000,C 90.000,E1 123.420} C_DIS
LIN {X 0.131,Y -325.092,Z 1246.684,A 0.000,B 0.000,C 90.000,E1 123.086} C_DIS
LIN {X -0.088,Y -338.239,Z 1246.665,A 0.000,B 0.000,C 90.000,E1 119.667} C_DIS
LIN {X 0.054,Y -350.402,Z 1246.649,A 0.000,B 0.000,C 90.000,E1 116.873} C_DIS
LIN {X 0.091,Y -364.038,Z 1246.634,A 0.000,B 0.000,C 90.000,E1 114.155} C_DIS
LIN {X -0.232,Y -377.498,Z 1246.621,A 0.000,B 0.000,C 90.000,E1 111.844} C_DIS
LIN {X -0.026,Y -392.312,Z 1246.608,A 0.000,B 0.000,C 90.000,E1 109.504} C_DIS
LIN {X 0.172,Y -408.585,Z 1246.596,A 0.000,B 0.000,C 90.000,E1 107.221} C_DIS
LIN {X -0.135,Y -426.432,Z 1246.584,A 0.000,B 0.000,C 90.000,E1 105.064} C_DIS
LIN {X -0.163,Y -445.866,Z 1246.572,A 0.000,B 0.000,C 90.000,E1 102.939} C_DIS
LIN {X -0.045,Y -466.086,Z 1246.561,A 0.000,B 0.000,C 90.000,E1 100.950} C_DIS
LIN {X -0.064,Y -473.793,Z 1246.557,A 0.000,B 0.000,C 90.000,E1 100.254} C_DIS
LIN {X -0.029,Y -475.867,Z 1246.556,A 0.000,B 0.000,C 90.000,E1 100.018} C_DIS
LIN {X -0.074,Y -477.444,Z 1246.554,A 0.000,B 0.000,C 90.000,E1 99.792} C_DIS
LIN {X -0.205,Y -478.746,Z 1246.553,A 0.000,B 0.000,C 90.000,E1 99.557} C_DIS
LIN {X 0.138,Y -479.705,Z 1246.552,A 0.000,B 0.000,C 90.000,E1 99.265} C_DIS
LIN {X -0.186,Y -480.772,Z 1246.549,A 0.000,B 0.000,C 90.000,E1 98.803} C_DIS
LIN {X 0.042,Y -480.841,Z 1246.546,A 0.000,B 0.000,C 90.000,E1 98.276} C_DIS
LIN {X 0.207,Y -479.927,Z 1246.543,A 0.000,B 0.000,C 90.000,E1 97.757} C_DIS
LIN {X -0.103,Y -477.873,Z 1246.540,A 0.000,B 0.000,C 90.000,E1 97.296} C_DIS
LIN {X 0.184,Y -476.286,Z 1246.539,A 0.000,B 0.000,C 90.000,E1 97.011} C_DIS
LIN {X 0.022,Y -456.179,Z 1246.524,A 0.000,B 0.000,C 90.000,E1 94.245} C_DIS
LIN {X -0.200,Y -435.665,Z 1246.506,A 0.000,B 0.000,C 90.000,E1 91.146} C_DIS
LIN {X 0.049,Y -418.757,Z 1246.490,A 0.000,B 0.000,C 90.000,E1 88.165} C_DIS
LIN {X 0.064,Y -405.933,Z 1246.476,A 0.000,B 0.000,C 90.000,E1 85.698} C_DIS
LIN {X 0.096,Y -395.772,Z 1246.465,A 0.000,B 0.000,C 90.000,E1 83.742} C_DIS
LIN {X -0.040,Y -385.537,Z 1246.454,A 0.000,B 0.000,C 90.000,E1 81.781} C_DIS
LIN {X 0.084,Y -376.552,Z 1246.445,A 0.000,B 0.000,C 90.000,E1 80.038} C_DIS
LIN {X 0.111,Y -367.263,Z 1246.435,A 0.000,B 0.000,C 90.000,E1 78.285} C_DIS
LIN {X 0.050,Y -357.701,Z 1246.425,A 0.000,B 0.000,C 90.000,E1 76.520} C_DIS
LIN {X 0.172,Y -346.267,Z 1246.413,A 0.000,B 0.000,C 90.000,E1 74.393} C_DIS
LIN {X 0.116,Y -333.368,Z 1246.400,A 0.000,B 0.000,C 90.000,E1 71.945} C_DIS
LIN {X 0.063,Y -320.810,Z 1246.386,A 0.000,B 0.000,C 90.000,E1 69.444} C_DIS
LIN {X -0.030,Y -304.704,Z 1246.366,A 0.000,B 0.000,C 90.000,E1 65.921} C_DIS
LIN {X -0.032,Y -290.141,Z 1246.346,A 0.000,B 0.000,C 90.000,E1 62.281} C_DIS
LIN {X 0.070,Y -278.141,Z 1246.327,A 0.000,B 0.000,C 90.000,E1 58.869} C_DIS
LIN {X 0.069,Y -268.220,Z 1246.310,A 0.000,B 0.000,C 90.000,E1 55.754} C_DIS
LIN {X -0.117,Y -258.085,Z 1246.290,A 0.000,B 0.000,C 90.000,E1 52.271} C_DIS
LIN {X -0.018,Y -250.660,Z 1246.274,A 0.000,B 0.000,C 90.000,E1 49.380} C_DIS
LIN {X 0.006,Y -241.916,Z 1246.254,A 0.000,B 0.000,C 90.000,E1 45.729} C_DIS
LIN {X -0.118,Y -236.912,Z 1246.242,A 0.000,B 0.000,C 90.000,E1 43.542} C_DIS
LIN {X -0.010,Y -228.784,Z 1246.221,A 0.000,B 0.000,C 90.000,E1 39.769} C_DIS
LIN {X -0.027,Y -221.186,Z 1246.200,A 0.000,B 0.000,C 90.000,E1 35.964} C_DIS
LIN {X 0.015,Y -214.306,Z 1246.178,A 0.000,B 0.000,C 90.000,E1 32.084} C_DIS
LIN {X 0.038,Y -208.276,Z 1246.156,A 0.000,B 0.000,C 90.000,E1 28.153} C_DIS
LIN {X -0.062,Y -203.139,Z 1246.134,A 0.000,B 0.000,C 90.000,E1 24.207} C_DIS
LIN {X -0.008,Y -198.824,Z 1246.112,A 0.000,B 0.000,C 90.000,E1 20.174} C_DIS
LIN {X -0.059,Y -195.289,Z 1246.090,A 0.000,B 0.000,C 90.000,E1 16.134} C_DIS
LIN {X 0.083,Y -191.792,Z 1246.058,A 0.000,B 0.000,C 90.000,E1 10.366} C_DIS
LIN {X -0.012,Y -191.637,Z 1245.974,A 0.000,B 0.000,C 90.000,E1 355.412} C_DIS
LIN {X -0.101,Y -194.778,Z 1245.943,A 0.000,B 0.000,C 90.000,E1 349.690} C_DIS
LIN {X 0.048,Y -198.638,Z 1245.915,A 0.000,B 0.000,C 90.000,E1 344.755} C_DIS
LIN {X -0.019,Y -202.720,Z 1245.893,A 0.000,B 0.000,C 90.000,E1 340.732} C_DIS
LIN {X -0.073,Y -207.524,Z 1245.871,A 0.000,B 0.000,C 90.000,E1 336.741} C_DIS
LIN {X 0.058,Y -212.995,Z 1245.849,A 0.000,B 0.000,C 90.000,E1 332.743} C_DIS
LIN {X -0.099,Y -219.079,Z 1245.827,A 0.000,B 0.000,C 90.000,E1 328.869} C_DIS
LIN {X 0.017,Y -225.842,Z 1245.805,A 0.000,B 0.000,C 90.000,E1 324.975} C_DIS
LIN {X 0.003,Y -233.296,Z 1245.784,A 0.000,B 0.000,C 90.000,E1 321.170} C_DIS
LIN {X 0.130,Y -241.696,Z 1245.763,A 0.000,B 0.000,C 90.000,E1 317.391} C_DIS
LIN {X 0.150,Y -251.204,Z 1245.743,A 0.000,B 0.000,C 90.000,E1 313.704} C_DIS
LIN {X -0.103,Y -258.751,Z 1245.729,A 0.000,B 0.000,C 90.000,E1 311.229} C_DIS
LIN {X -0.024,Y -266.231,Z 1245.717,A 0.000,B 0.000,C 90.000,E1 309.072} C_DIS
LIN {X 0.038,Y -274.677,Z 1245.705,A 0.000,B 0.000,C 90.000,E1 306.950} C_DIS
LIN {X -0.071,Y -284.068,Z 1245.694,A 0.000,B 0.000,C 90.000,E1 304.898} C_DIS
LIN {X 0.062,Y -296.131,Z 1245.681,A 0.000,B 0.000,C 90.000,E1 302.498} C_DIS
LIN {X 0.007,Y -305.724,Z 1245.671,A 0.000,B 0.000,C 90.000,E1 300.846} C_DIS
LIN {X 0.041,Y -316.552,Z 1245.662,A 0.000,B 0.000,C 90.000,E1 299.205} C_DIS
LIN {X 0.112,Y -328.623,Z 1245.653,A 0.000,B 0.000,C 90.000,E1 297.590} C_DIS
LIN {X 0.037,Y -351.745,Z 1245.638,A 0.000,B 0.000,C 90.000,E1 294.823} C_DIS
LIN {X -0.143,Y -367.533,Z 1245.628,A 0.000,B 0.000,C 90.000,E1 293.078} C_DIS
LIN {X -0.018,Y -380.429,Z 1245.620,A 0.000,B 0.000,C 90.000,E1 291.642} C_DIS
LIN {X -0.221,Y -393.325,Z 1245.612,A 0.000,B 0.000,C 90.000,E1 290.248} C_DIS
LIN {X 0.106,Y -411.152,Z 1245.602,A 0.000,B 0.000,C 90.000,E1 288.308} C_DIS
LIN {X -0.104,Y -421.186,Z 1245.596,A 0.000,B 0.000,C 90.000,E1 287.275} C_DIS
LIN {X 0.074,Y -428.404,Z 1245.591,A 0.000,B 0.000,C 90.000,E1 286.441} C_DIS
LIN {X -0.135,Y -435.110,Z 1245.587,A 0.000,B 0.000,C 90.000,E1 285.662} C_DIS
LIN {X 0.127,Y -441.256,Z 1245.583,A 0.000,B 0.000,C 90.000,E1 284.828} C_DIS
LIN {X -0.087,Y -446.812,Z 1245.578,A 0.000,B 0.000,C 90.000,E1 284.064} C_DIS
LIN {X 0.182,Y -451.658,Z 1245.574,A 0.000,B 0.000,C 90.000,E1 283.244} C_DIS
LIN {X 0.063,Y -455.723,Z 1245.569,A 0.000,B 0.000,C 90.000,E1 282.479} C_DIS
LIN {X 0.151,Y -458.132,Z 1245.567,A 0.000,B 0.000,C 90.000,E1 281.951} C_DIS
LIN {X 0.082,Y -461.135,Z 1245.562,A 0.000,B 0.000,C 90.000,E1 281.186} C_DIS
LIN {X 0.195,Y -462.855,Z 1245.559,A 0.000,B 0.000,C 90.000,E1 280.658} C_DIS
LIN {X -0.222,Y -464.305,Z 1245.557,A 0.000,B 0.000,C 90.000,E1 280.197} C_DIS
LIN {X -0.090,Y -465.477,Z 1245.554,A 0.000,B 0.000,C 90.000,E1 279.670} C_DIS
LIN {X -0.027,Y -466.374,Z 1245.551,A 0.000,B 0.000,C 90.000,E1 279.151} C_DIS
LIN {X 0.117,Y -467.009,Z 1245.548,A 0.000,B 0.000,C 90.000,E1 278.624} C_DIS
LIN {X 0.194,Y -467.339,Z 1245.545,A 0.000,B 0.000,C 90.000,E1 278.106} C_DIS
LIN {X -0.184,Y -467.306,Z 1245.542,A 0.000,B 0.000,C 90.000,E1 277.644} C_DIS
LIN {X -0.098,Y -466.844,Z 1245.540,A 0.000,B 0.000,C 90.000,E1 277.125} C_DIS
LIN {X -0.010,Y -465.934,Z 1245.537,A 0.000,B 0.000,C 90.000,E1 276.606} C_DIS
LIN {X 0.074,Y -464.533,Z 1245.534,A 0.000,B 0.000,C 90.000,E1 276.087} C_DIS
LIN {X 0.153,Y -462.735,Z 1245.531,A 0.000,B 0.000,C 90.000,E1 275.568} C_DIS
LIN {X 0.222,Y -460.535,Z 1245.528,A 0.000,B 0.000,C 90.000,E1 275.049} C_DIS
LIN {X -0.185,Y -457.907,Z 1245.525,A 0.000,B 0.000,C 90.000,E1 274.588} C_DIS
LIN {X -0.149,Y -454.719,Z 1245.522,A 0.000,B 0.000,C 90.000,E1 274.069} C_DIS
LIN {X -0.160,Y -450.670,Z 1245.520,A 0.000,B 0.000,C 90.000,E1 273.555} C_DIS
LIN {X 0.050,Y -448.260,Z 1245.518,A 0.000,B 0.000,C 90.000,E1 273.269} C_DIS
LIN {X -0.163,Y -445.532,Z 1245.517,A 0.000,B 0.000,C 90.000,E1 273.037} C_DIS
LIN {X 0.042,Y -439.426,Z 1245.514,A 0.000,B 0.000,C 90.000,E1 272.522} C_DIS
LIN {X -0.108,Y -432.709,Z 1245.512,A 0.000,B 0.000,C 90.000,E1 272.121} C_DIS
LIN {X -0.149,Y -425.610,Z 1245.510,A 0.000,B 0.000,C 90.000,E1 271.776} C_DIS
LIN {X -0.126,Y -418.559,Z 1245.508,A 0.000,B 0.000,C 90.000,E1 271.489} C_DIS
LIN {X -0.161,Y -411.623,Z 1245.507,A 0.000,B 0.000,C 90.000,E1 271.260} C_DIS
LIN {X -0.168,Y -400.875,Z 1245.505,A 0.000,B 0.000,C 90.000,E1 270.974} C_DIS
LIN {X -0.122,Y -389.298,Z 1245.504,A 0.000,B 0.000,C 90.000,E1 270.745} C_DIS
LIN {X -0.123,Y -380.740,Z 1245.503,A 0.000,B 0.000,C 90.000,E1 270.630} C_DIS
LIN {X 0.175,Y -372.795,Z 1245.503,A 0.000,B 0.000,C 90.000,E1 270.516} C_DIS
LIN {X -0.022,Y -363.832,Z 1245.503,A 0.000,B 0.000,C 90.000,E1 270.516} C_DIS
LIN {X -0.035,Y -181.564,Z 1245.503,A 0.000,B 0.000,C 90.000,E1 270.516} C_DIS
LIN {X -0.003,Y -181.114,Z 1245.489,A 0.000,B 0.000,C 90.000,E1 267.936} C_DIS
LIN {X -0.014,Y -180.907,Z 1245.474,A 0.000,B 0.000,C 90.000,E1 265.412} C_DIS
LIN {X 0.041,Y -180.708,Z 1245.470,A 0.000,B 0.000,C 90.000,E1 264.552} C_DIS
LIN {X -0.040,Y -178.794,Z 1245.442,A 0.000,B 0.000,C 90.000,E1 259.511} C_DIS
LIN {X 0.037,Y -175.839,Z 1245.413,A 0.000,B 0.000,C 90.000,E1 254.393} C_DIS
LIN {X 0.037,Y -172.030,Z 1245.385,A 0.000,B 0.000,C 90.000,E1 249.263} C_DIS
LIN {X 0.013,Y -171.458,Z 1245.380,A 0.000,B 0.000,C 90.000,E1 248.411} C_DIS
LIN {X -0.006,Y -167.691,Z 1245.356,A 0.000,B 0.000,C 90.000,E1 244.101} C_DIS
LIN {X 0.007,Y -166.372,Z 1245.346,A 0.000,B 0.000,C 90.000,E1 242.359} C_DIS
LIN {X -0.001,Y -163.102,Z 1245.327,A 0.000,B 0.000,C 90.000,E1 238.869} C_DIS
LIN {X 0.050,Y -161.048,Z 1245.312,A 0.000,B 0.000,C 90.000,E1 236.215} C_DIS
LIN {X 0.033,Y -157.785,Z 1245.293,A 0.000,B 0.000,C 90.000,E1 232.683} C_DIS
LIN {X -0.024,Y -155.822,Z 1245.278,A 0.000,B 0.000,C 90.000,E1 230.033} C_DIS
LIN {X -0.066,Y -152.073,Z 1245.253,A 0.000,B 0.000,C 90.000,E1 225.567} C_DIS
LIN {X -0.047,Y -150.323,Z 1245.238,A 0.000,B 0.000,C 90.000,E1 222.852} C_DIS
LIN {X -0.025,Y -147.065,Z 1245.213,A 0.000,B 0.000,C 90.000,E1 218.302} C_DIS
LIN {X 0.081,Y -145.641,Z 1245.198,A 0.000,B 0.000,C 90.000,E1 215.518} C_DIS
LIN {X 0.080,Y -143.023,Z 1245.172,A 0.000,B 0.000,C 90.000,E1 210.924} C_DIS
LIN {X 0.011,Y -141.649,Z 1245.151,A 0.000,B 0.000,C 90.000,E1 207.257} C_DIS
LIN {X 0.061,Y -139.442,Z 1245.115,A 0.000,B 0.000,C 90.000,E1 200.737} C_DIS
LIN {X -0.017,Y -139.176,Z 1245.105,A 0.000,B 0.000,C 90.000,E1 198.906} C_DIS
LIN {X 0.011,Y -138.318,Z 1245.053,A 0.000,B 0.000,C 90.000,E1 189.557} C_DIS
LIN {X 0.020,Y -139.469,Z 1245.006,A 0.000,B 0.000,C 90.000,E1 181.146} C_DIS
LIN {X -0.039,Y -141.038,Z 1244.975,A 0.000,B 0.000,C 90.000,E1 175.584} C_DIS
LIN {X 0.056,Y -142.406,Z 1244.960,A 0.000,B 0.000,C 90.000,E1 172.761} C_DIS
LIN {X -0.023,Y -144.639,Z 1244.934,A 0.000,B 0.000,C 90.000,E1 168.173} C_DIS
LIN {X 0.036,Y -147.835,Z 1244.909,A 0.000,B 0.000,C 90.000,E1 163.559} C_DIS
LIN {X -0.019,Y -150.530,Z 1244.888,A 0.000,B 0.000,C 90.000,E1 159.934} C_DIS
LIN {X 0.000,Y -153.994,Z 1244.868,A 0.000,B 0.000,C 90.000,E1 156.305} C_DIS
LIN {X -0.079,Y -157.407,Z 1244.848,A 0.000,B 0.000,C 90.000,E1 152.743} C_DIS
LIN {X 0.000,Y -161.615,Z 1244.829,A 0.000,B 0.000,C 90.000,E1 149.154} C_DIS
LIN {X 0.102,Y -165.812,Z 1244.809,A 0.000,B 0.000,C 90.000,E1 145.595} C_DIS
LIN {X -0.010,Y -170.780,Z 1244.790,A 0.000,B 0.000,C 90.000,E1 142.145} C_DIS
LIN {X 0.012,Y -175.650,Z 1244.771,A 0.000,B 0.000,C 90.000,E1 138.690} C_DIS
LIN {X 0.010,Y -181.265,Z 1244.752,A 0.000,B 0.000,C 90.000,E1 135.283} C_DIS
LIN {X 0.011,Y -186.739,Z 1244.733,A 0.000,B 0.000,C 90.000,E1 131.919} C_DIS
LIN {X -0.038,Y -191.336,Z 1244.719,A 0.000,B 0.000,C 90.000,E1 129.439} C_DIS
LIN {X 0.008,Y -197.170,Z 1244.701,A 0.000,B 0.000,C 90.000,E1 126.137} C_DIS
LIN {X 0.012,Y -200.556,Z 1244.691,A 0.000,B 0.000,C 90.000,E1 124.452} C_DIS
LIN {X -0.034,Y -310.222,Z 1244.691,A 0.000,B 0.000,C 90.000,E1 124.452} C_DIS
LIN {X -0.100,Y -315.780,Z 1244.690,A 0.000,B 0.000,C 90.000,E1 124.278} C_DIS
LIN {X 0.012,Y -318.295,Z 1244.689,A 0.000,B 0.000,C 90.000,E1 124.072} C_DIS
LIN {X -0.025,Y -321.647,Z 1244.687,A 0.000,B 0.000,C 90.000,E1 123.706} C_DIS
LIN {X 0.155,Y -323.582,Z 1244.686,A 0.000,B 0.000,C 90.000,E1 123.372} C_DIS
LIN {X 0.064,Y -325.096,Z 1244.684,A 0.000,B 0.000,C 90.000,E1 123.086} C_DIS
LIN {X -0.156,Y -330.921,Z 1244.675,A 0.000,B 0.000,C 90.000,E1 121.544} C_DIS
LIN {X 0.105,Y -342.164,Z 1244.660,A 0.000,B 0.000,C 90.000,E1 118.693} C_DIS
LIN {X -0.100,Y -354.810,Z 1244.644,A 0.000,B 0.000,C 90.000,E1 115.976} C_DIS
LIN {X 0.048,Y -368.975,Z 1244.629,A 0.000,B 0.000,C 90.000,E1 113.259} C_DIS
LIN {X 0.047,Y -382.937,Z 1244.616,A 0.000,B 0.000,C 90.000,E1 110.918} C_DIS
LIN {X -0.110,Y -398.293,Z 1244.604,A 0.000,B 0.000,C 90.000,E1 108.652} C_DIS
LIN {X 0.116,Y -415.150,Z 1244.591,A 0.000,B 0.000,C 90.000,E1 106.386} C_DIS
LIN {X -0.145,Y -433.629,Z 1244.579,A 0.000,B 0.000,C 90.000,E1 104.245} C_DIS
LIN {X 0.222,Y -453.468,Z 1244.568,A 0.000,B 0.000,C 90.000,E1 102.119} C_DIS
LIN {X -0.141,Y -473.850,Z 1244.557,A 0.000,B 0.000,C 90.000,E1 100.254} C_DIS
LIN {X -0.114,Y -475.885,Z 1244.556,A 0.000,B 0.000,C 90.000,E1 100.018} C_DIS
LIN {X -0.169,Y -477.433,Z 1244.554,A 0.000,B 0.000,C 90.000,E1 99.792} C_DIS
LIN {X 0.173,Y -478.705,Z 1244.553,A 0.000,B 0.000,C 90.000,E1 99.500} C_DIS
LIN {X 0.043,Y -479.639,Z 1244.552,A 0.000,B 0.000,C 90.000,E1 99.265} C_DIS
LIN {X 0.194,Y -480.664,Z 1244.549,A 0.000,B 0.000,C 90.000,E1 98.746} C_DIS
LIN {X -0.053,Y -480.695,Z 1244.546,A 0.000,B 0.000,C 90.000,E1 98.276} C_DIS
LIN {X 0.110,Y -479.740,Z 1244.543,A 0.000,B 0.000,C 90.000,E1 97.757} C_DIS
LIN {X -0.199,Y -477.635,Z 1244.540,A 0.000,B 0.000,C 90.000,E1 97.296} C_DIS
LIN {X 0.087,Y -476.013,Z 1244.539,A 0.000,B 0.000,C 90.000,E1 97.011} C_DIS
LIN {X 0.143,Y -457.694,Z 1244.525,A 0.000,B 0.000,C 90.000,E1 94.473} C_DIS
LIN {X 0.131,Y -435.405,Z 1244.506,A 0.000,B 0.000,C 90.000,E1 91.088} C_DIS
LIN {X -0.059,Y -418.511,Z 1244.490,A 0.000,B 0.000,C 90.000,E1 88.165} C_DIS
LIN {X -0.048,Y -405.687,Z 1244.476,A 0.000,B 0.000,C 90.000,E1 85.698} C_DIS
LIN {X -0.018,Y -395.514,Z 1244.465,A 0.000,B 0.000,C 90.000,E1 83.742} C_DIS
LIN {X -0.156,Y -385.283,Z 1244.454,A 0.000,B 0.000,C 90.000,E1 81.781} C_DIS
LIN {X -0.035,Y -376.309,Z 1244.445,A 0.000,B 0.000,C 90.000,E1 80.038} C_DIS
LIN {X -0.009,Y -367.007,Z 1244.435,A 0.000,B 0.000,C 90.000,E1 78.285} C_DIS
LIN {X -0.071,Y -357.470,Z 1244.425,A 0.000,B 0.000,C 90.000,E1 76.520} C_DIS
LIN {X 0.033,Y -347.686,Z 1244.415,A 0.000,B 0.000,C 90.000,E1 74.700} C_DIS
LIN {X 0.111,Y -334.746,Z 1244.401,A 0.000,B 0.000,C 90.000,E1 72.236} C_DIS
LIN {X -0.011,Y -322.168,Z 1244.387,A 0.000,B 0.000,C 90.000,E1 69.752} C_DIS
LIN {X -0.062,Y -305.912,Z 1244.368,A 0.000,B 0.000,C 90.000,E1 66.230} C_DIS
LIN {X -0.147,Y -291.215,Z 1244.348,A 0.000,B 0.000,C 90.000,E1 62.615} C_DIS
LIN {X -0.011,Y -279.087,Z 1244.329,A 0.000,B 0.000,C 90.000,E1 59.203} C_DIS
LIN {X 0.087,Y -267.961,Z 1244.310,A 0.000,B 0.000,C 90.000,E1 55.722} C_DIS
LIN {X 0.108,Y -257.801,Z 1244.290,A 0.000,B 0.000,C 90.000,E1 52.190} C_DIS
LIN {X 0.033,Y -250.361,Z 1244.274,A 0.000,B 0.000,C 90.000,E1 49.337} C_DIS
LIN {X -0.137,Y -241.590,Z 1244.254,A 0.000,B 0.000,C 90.000,E1 45.729} C_DIS
LIN {X 0.070,Y -236.553,Z 1244.242,A 0.000,B 0.000,C 90.000,E1 43.461} C_DIS
LIN {X 0.013,Y -228.386,Z 1244.221,A 0.000,B 0.000,C 90.000,E1 39.725} C_DIS
LIN {X -0.056,Y -220.753,Z 1244.200,A 0.000,B 0.000,C 90.000,E1 35.931} C_DIS
LIN {X -0.040,Y -213.848,Z 1244.178,A 0.000,B 0.000,C 90.000,E1 32.054} C_DIS
LIN {X 0.044,Y -207.834,Z 1244.156,A 0.000,B 0.000,C 90.000,E1 28.103} C_DIS
LIN {X 0.019,Y -202.675,Z 1244.134,A 0.000,B 0.000,C 90.000,E1 24.131} C_DIS
LIN {X -0.019,Y -198.379,Z 1244.112,A 0.000,B 0.000,C 90.000,E1 20.120} C_DIS
LIN {X -0.079,Y -194.864,Z 1244.089,A 0.000,B 0.000,C 90.000,E1 16.079} C_DIS
LIN {X 0.051,Y -191.422,Z 1244.057,A 0.000,B 0.000,C 90.000,E1 10.310} C_DIS
LIN {X -0.021,Y -191.370,Z 1243.974,A 0.000,B 0.000,C 90.000,E1 355.412} C_DIS
LIN {X 0.071,Y -194.535,Z 1243.943,A 0.000,B 0.000,C 90.000,E1 349.634} C_DIS
LIN {X 0.018,Y -198.403,Z 1243.915,A 0.000,B 0.000,C 90.000,E1 344.755} C_DIS
LIN {X -0.057,Y -202.514,Z 1243.893,A 0.000,B 0.000,C 90.000,E1 340.732} C_DIS
LIN {X -0.118,Y -207.356,Z 1243.871,A 0.000,B 0.000,C 90.000,E1 336.741} C_DIS
LIN {X 0.007,Y -212.858,Z 1243.849,A 0.000,B 0.000,C 90.000,E1 332.743} C_DIS
LIN {X 0.032,Y -218.961,Z 1243.827,A 0.000,B 0.000,C 90.000,E1 328.820} C_DIS
LIN {X -0.044,Y -225.737,Z 1243.805,A 0.000,B 0.000,C 90.000,E1 324.975} C_DIS
LIN {X -0.064,Y -233.193,Z 1243.784,A 0.000,B 0.000,C 90.000,E1 321.170} C_DIS
LIN {X 0.058,Y -241.605,Z 1243.763,A 0.000,B 0.000,C 90.000,E1 317.391} C_DIS
LIN {X -0.101,Y -250.113,Z 1243.745,A 0.000,B 0.000,C 90.000,E1 314.109} C_DIS
LIN {X -0.015,Y -258.700,Z 1243.729,A 0.000,B 0.000,C 90.000,E1 311.191} C_DIS
LIN {X 0.057,Y -266.188,Z 1243.717,A 0.000,B 0.000,C 90.000,E1 309.036} C_DIS
LIN {X 0.035,Y -276.154,Z 1243.703,A 0.000,B 0.000,C 90.000,E1 306.583} C_DIS
LIN {X 0.040,Y -289.022,Z 1243.688,A 0.000,B 0.000,C 90.000,E1 303.833} C_DIS
LIN {X 0.121,Y -299.796,Z 1243.677,A 0.000,B 0.000,C 90.000,E1 301.799} C_DIS
LIN {X -0.074,Y -307.711,Z 1243.669,A 0.000,B 0.000,C 90.000,E1 300.512} C_DIS
LIN {X -0.066,Y -316.443,Z 1243.662,A 0.000,B 0.000,C 90.000,E1 299.205} C_DIS
LIN {X 0.093,Y -331.055,Z 1243.651,A 0.000,B 0.000,C 90.000,E1 297.257} C_DIS
LIN {X 0.078,Y -351.466,Z 1243.638,A 0.000,B 0.000,C 90.000,E1 294.823} C_DIS
LIN {X 0.135,Y -369.756,Z 1243.627,A 0.000,B 0.000,C 90.000,E1 292.770} C_DIS
LIN {X 0.076,Y -382.720,Z 1243.619,A 0.000,B 0.000,C 90.000,E1 291.354} C_DIS
LIN {X -0.118,Y -398.252,Z 1243.609,A 0.000,B 0.000,C 90.000,E1 289.685} C_DIS
LIN {X 0.054,Y -411.147,Z 1243.602,A 0.000,B 0.000,C 90.000,E1 288.308} C_DIS
LIN {X -0.196,Y -421.231,Z 1243.596,A 0.000,B 0.000,C 90.000,E1 287.275} C_DIS
LIN {X -0.024,Y -428.455,Z 1243.591,A 0.000,B 0.000,C 90.000,E1 286.441} C_DIS
LIN {X 0.185,Y -435.144,Z 1243.587,A 0.000,B 0.000,C 90.000,E1 285.607} C_DIS
LIN {X 0.028,Y -441.275,Z 1243.582,A 0.000,B 0.000,C 90.000,E1 284.828} C_DIS
LIN {X -0.187,Y -446.855,Z 1243.578,A 0.000,B 0.000,C 90.000,E1 284.064} C_DIS
LIN {X 0.081,Y -451.687,Z 1243.574,A 0.000,B 0.000,C 90.000,E1 283.244} C_DIS
LIN {X -0.038,Y -455.795,Z 1243.569,A 0.000,B 0.000,C 90.000,E1 282.479} C_DIS
LIN {X -0.128,Y -459.202,Z 1243.565,A 0.000,B 0.000,C 90.000,E1 281.715} C_DIS
LIN {X -0.020,Y -461.170,Z 1243.562,A 0.000,B 0.000,C 90.000,E1 281.186} C_DIS
LIN {X 0.092,Y -462.878,Z 1243.559,A 0.000,B 0.000,C 90.000,E1 280.658} C_DIS
LIN {X 0.133,Y -464.325,Z 1243.556,A 0.000,B 0.000,C 90.000,E1 280.141} C_DIS
LIN {X -0.192,Y -465.518,Z 1243.554,A 0.000,B 0.000,C 90.000,E1 279.670} C_DIS
LIN {X -0.130,Y -466.413,Z 1243.551,A 0.000,B 0.000,C 90.000,E1 279.151} C_DIS
LIN {X 0.014,Y -467.066,Z 1243.548,A 0.000,B 0.000,C 90.000,E1 278.624} C_DIS
LIN {X 0.092,Y -467.406,Z 1243.545,A 0.000,B 0.000,C 90.000,E1 278.106} C_DIS
LIN {X 0.176,Y -467.385,Z 1243.542,A 0.000,B 0.000,C 90.000,E1 277.587} C_DIS
LIN {X -0.200,Y -466.911,Z 1243.539,A 0.000,B 0.000,C 90.000,E1 277.125} C_DIS
LIN {X -0.112,Y -466.022,Z 1243.537,A 0.000,B 0.000,C 90.000,E1 276.606} C_DIS
LIN {X -0.026,Y -464.670,Z 1243.534,A 0.000,B 0.000,C 90.000,E1 276.087} C_DIS
LIN {X 0.054,Y -462.880,Z 1243.531,A 0.000,B 0.000,C 90.000,E1 275.568} C_DIS
LIN {X -0.098,Y -459.463,Z 1243.527,A 0.000,B 0.000,C 90.000,E1 274.821} C_DIS
LIN {X -0.052,Y -456.562,Z 1243.524,A 0.000,B 0.000,C 90.000,E1 274.302} C_DIS
LIN {X -0.023,Y -452.928,Z 1243.521,A 0.000,B 0.000,C 90.000,E1 273.784} C_DIS
LIN {X 0.197,Y -450.813,Z 1243.520,A 0.000,B 0.000,C 90.000,E1 273.498} C_DIS
LIN {X 0.190,Y -445.691,Z 1243.517,A 0.000,B 0.000,C 90.000,E1 272.980} C_DIS
LIN {X -0.081,Y -439.541,Z 1243.514,A 0.000,B 0.000,C 90.000,E1 272.522} C_DIS
LIN {X 0.182,Y -432.758,Z 1243.512,A 0.000,B 0.000,C 90.000,E1 272.064} C_DIS
LIN {X 0.181,Y -425.804,Z 1243.510,A 0.000,B 0.000,C 90.000,E1 271.718} C_DIS
LIN {X 0.195,Y -418.706,Z 1243.508,A 0.000,B 0.000,C 90.000,E1 271.432} C_DIS
LIN {X 0.179,Y -411.941,Z 1243.507,A 0.000,B 0.000,C 90.000,E1 271.203} C_DIS
LIN {X 0.186,Y -401.378,Z 1243.505,A 0.000,B 0.000,C 90.000,E1 270.917} C_DIS
LIN {X -0.081,Y -393.999,Z 1243.504,A 0.000,B 0.000,C 90.000,E1 270.802} C_DIS
LIN {X -0.149,Y -382.039,Z 1243.503,A 0.000,B 0.000,C 90.000,E1 270.630} C_DIS
LIN {X -0.027,Y -370.788,Z 1243.503,A 0.000,B 0.000,C 90.000,E1 270.516} C_DIS
LIN {X -0.132,Y -364.905,Z 1243.503,A 0.000,B 0.000,C 90.000,E1 270.516} C_DIS
LIN {X 0.090,Y -181.567,Z 1243.503,A 0.000,B 0.000,C 90.000,E1 270.458} C_DIS
LIN {X -0.050,Y -181.111,Z 1243.488,A 0.000,B 0.000,C 90.000,E1 267.936} C_DIS
LIN {X -0.062,Y -180.907,Z 1243.474,A 0.000,B 0.000,C 90.000,E1 265.412} C_DIS
LIN {X 0.012,Y -180.701,Z 1243.470,A 0.000,B 0.000,C 90.000,E1 264.546} C_DIS
LIN {X 0.090,Y -178.785,Z 1243.442,A 0.000,B 0.000,C 90.000,E1 259.454} C_DIS
LIN {X -0.008,Y -175.832,Z 1243.413,A 0.000,B 0.000,C 90.000,E1 254.393} C_DIS
LIN {X -0.008,Y -172.021,Z 1243.385,A 0.000,B 0.000,C 90.000,E1 249.263} C_DIS
LIN {X -0.032,Y -171.445,Z 1243.380,A 0.000,B 0.000,C 90.000,E1 248.411} C_DIS
LIN {X 0.022,Y -167.679,Z 1243.356,A 0.000,B 0.000,C 90.000,E1 244.076} C_DIS
LIN {X -0.037,Y -166.356,Z 1243.346,A 0.000,B 0.000,C 90.000,E1 242.359} C_DIS
LIN {X -0.044,Y -163.089,Z 1243.327,A 0.000,B 0.000,C 90.000,E1 238.869} C_DIS
LIN {X 0.006,Y -161.033,Z 1243.312,A 0.000,B 0.000,C 90.000,E1 236.215} C_DIS
LIN {X -0.010,Y -157.772,Z 1243.293,A 0.000,B 0.000,C 90.000,E1 232.683} C_DIS
LIN {X 0.053,Y -155.810,Z 1243.278,A 0.000,B 0.000,C 90.000,E1 229.989} C_DIS
LIN {X 0.000,Y -152.061,Z 1243.253,A 0.000,B 0.000,C 90.000,E1 225.526} C_DIS
LIN {X 0.014,Y -150.312,Z 1243.238,A 0.000,B 0.000,C 90.000,E1 222.813} C_DIS
LIN {X 0.050,Y -147.055,Z 1243.213,A 0.000,B 0.000,C 90.000,E1 218.257} C_DIS
LIN {X 0.041,Y -145.633,Z 1243.197,A 0.000,B 0.000,C 90.000,E1 215.518} C_DIS
LIN {X 0.040,Y -143.016,Z 1243.172,A 0.000,B 0.000,C 90.000,E1 210.924} C_DIS
LIN {X -0.030,Y -141.642,Z 1243.151,A 0.000,B 0.000,C 90.000,E1 207.257} C_DIS
LIN {X 0.021,Y -139.440,Z 1243.115,A 0.000,B 0.000,C 90.000,E1 200.737} C_DIS
LIN {X -0.057,Y -139.173,Z 1243.105,A 0.000,B 0.000,C 90.000,E1 198.906} C_DIS
LIN {X -0.029,Y -138.318,Z 1243.053,A 0.000,B 0.000,C 90.000,E1 189.557} C_DIS
LIN {X -0.019,Y -139.472,Z 1243.006,A 0.000,B 0.000,C 90.000,E1 181.146} C_DIS
LIN {X 0.061,Y -141.045,Z 1242.975,A 0.000,B 0.000,C 90.000,E1 175.527} C_DIS
LIN {X 0.016,Y -142.414,Z 1242.960,A 0.000,B 0.000,C 90.000,E1 172.761} C_DIS
LIN {X -0.064,Y -144.649,Z 1242.934,A 0.000,B 0.000,C 90.000,E1 168.173} C_DIS
LIN {X -0.004,Y -147.845,Z 1242.909,A 0.000,B 0.000,C 90.000,E1 163.559} C_DIS
LIN {X -0.061,Y -150.544,Z 1242.888,A 0.000,B 0.000,C 90.000,E1 159.934} C_DIS
LIN {X -0.042,Y -154.010,Z 1242.868,A 0.000,B 0.000,C 90.000,E1 156.305} C_DIS
LIN {X 0.017,Y -157.424,Z 1242.848,A 0.000,B 0.000,C 90.000,E1 152.692} C_DIS
LIN {X 0.039,Y -161.636,Z 1242.828,A 0.000,B 0.000,C 90.000,E1 149.125} C_DIS
LIN {X 0.057,Y -165.832,Z 1242.809,A 0.000,B 0.000,C 90.000,E1 145.595} C_DIS
LIN {X 0.050,Y -170.803,Z 1242.790,A 0.000,B 0.000,C 90.000,E1 142.110} C_DIS
LIN {X -0.034,Y -175.674,Z 1242.770,A 0.000,B 0.000,C 90.000,E1 138.690} C_DIS
LIN {X 0.091,Y -181.287,Z 1242.751,A 0.000,B 0.000,C 90.000,E1 135.243} C_DIS
LIN {X -0.037,Y -186.766,Z 1242.733,A 0.000,B 0.000,C 90.000,E1 131.919} C_DIS
LIN {X 0.035,Y -191.359,Z 1242.719,A 0.000,B 0.000,C 90.000,E1 129.402} C_DIS
LIN {X -0.041,Y -197.197,Z 1242.701,A 0.000,B 0.000,C 90.000,E1 126.137} C_DIS
LIN {X 0.071,Y -200.614,Z 1242.691,A 0.000,B 0.000,C 90.000,E1 124.405} C_DIS
LIN {X 0.074,Y -309.701,Z 1242.691,A 0.000,B 0.000,C 90.000,E1 124.405} C_DIS
LIN {X -0.203,Y -312.812,Z 1242.691,A 0.000,B 0.000,C 90.000,E1 124.405} C_DIS
LIN {X -0.066,Y -318.558,Z 1242.689,A 0.000,B 0.000,C 90.000,E1 124.040} C_DIS
LIN {X -0.104,Y -321.616,Z 1242.687,A 0.000,B 0.000,C 90.000,E1 123.706} C_DIS
LIN {X 0.072,Y -323.581,Z 1242.685,A 0.000,B 0.000,C 90.000,E1 123.372} C_DIS
LIN {X -0.022,Y -325.114,Z 1242.684,A 0.000,B 0.000,C 90.000,E1 123.086} C_DIS
LIN {X 0.099,Y -329.790,Z 1242.677,A 0.000,B 0.000,C 90.000,E1 121.799} C_DIS
LIN {X 0.036,Y -340.887,Z 1242.661,A 0.000,B 0.000,C 90.000,E1 118.999} C_DIS
LIN {X 0.094,Y -353.383,Z 1242.646,A 0.000,B 0.000,C 90.000,E1 116.232} C_DIS
LIN {X -0.120,Y -367.377,Z 1242.631,A 0.000,B 0.000,C 90.000,E1 113.567} C_DIS
LIN {X -0.170,Y -381.180,Z 1242.618,A 0.000,B 0.000,C 90.000,E1 111.227} C_DIS
LIN {X -0.001,Y -396.364,Z 1242.605,A 0.000,B 0.000,C 90.000,E1 108.906} C_DIS
LIN {X -0.087,Y -413.036,Z 1242.593,A 0.000,B 0.000,C 90.000,E1 106.677} C_DIS
LIN {X 0.003,Y -431.314,Z 1242.580,A 0.000,B 0.000,C 90.000,E1 104.481} C_DIS
LIN {X 0.244,Y -451.039,Z 1242.569,A 0.000,B 0.000,C 90.000,E1 102.355} C_DIS
LIN {X -0.238,Y -473.924,Z 1242.557,A 0.000,B 0.000,C 90.000,E1 100.254} C_DIS
LIN {X 0.245,Y -475.918,Z 1242.556,A 0.000,B 0.000,C 90.000,E1 99.962} C_DIS
LIN {X 0.259,Y -477.437,Z 1242.554,A 0.000,B 0.000,C 90.000,E1 99.726} C_DIS
LIN {X 0.050,Y -478.674,Z 1242.553,A 0.000,B 0.000,C 90.000,E1 99.500} C_DIS
LIN {X -0.081,Y -479.579,Z 1242.551,A 0.000,B 0.000,C 90.000,E1 99.265} C_DIS
LIN {X 0.070,Y -480.556,Z 1242.549,A 0.000,B 0.000,C 90.000,E1 98.746} C_DIS
LIN {X -0.177,Y -480.543,Z 1242.546,A 0.000,B 0.000,C 90.000,E1 98.276} C_DIS
LIN {X -0.014,Y -479.541,Z 1242.543,A 0.000,B 0.000,C 90.000,E1 97.757} C_DIS
LIN {X -0.201,Y -478.623,Z 1242.542,A 0.000,B 0.000,C 90.000,E1 97.530} C_DIS
LIN {X 0.149,Y -477.375,Z 1242.540,A 0.000,B 0.000,C 90.000,E1 97.239} C_DIS
LIN {X 0.018,Y -475.705,Z 1242.539,A 0.000,B 0.000,C 90.000,E1 97.004} C_DIS
LIN {X 0.010,Y -457.406,Z 1242.525,A 0.000,B 0.000,C 90.000,E1 94.473} C_DIS
LIN {X -0.176,Y -436.752,Z 1242.508,A 0.000,B 0.000,C 90.000,E1 91.375} C_DIS
LIN {X -0.140,Y -422.690,Z 1242.494,A 0.000,B 0.000,C 90.000,E1 88.969} C_DIS
LIN {X 0.145,Y -406.836,Z 1242.478,A 0.000,B 0.000,C 90.000,E1 85.927} C_DIS
LIN {X 0.128,Y -398.144,Z 1242.468,A 0.000,B 0.000,C 90.000,E1 84.261} C_DIS
LIN {X 0.041,Y -387.952,Z 1242.457,A 0.000,B 0.000,C 90.000,E1 82.299} C_DIS
LIN {X 0.148,Y -379.056,Z 1242.448,A 0.000,B 0.000,C 90.000,E1 80.566} C_DIS
LIN {X -0.149,Y -369.873,Z 1242.438,A 0.000,B 0.000,C 90.000,E1 78.870} C_DIS
LIN {X 0.115,Y -360.430,Z 1242.428,A 0.000,B 0.000,C 90.000,E1 77.061} C_DIS
LIN {X 0.012,Y -350.705,Z 1242.418,A 0.000,B 0.000,C 90.000,E1 75.283} C_DIS
LIN {X -0.026,Y -337.687,Z 1242.405,A 0.000,B 0.000,C 90.000,E1 72.851} C_DIS
LIN {X -0.082,Y -325.047,Z 1242.391,A 0.000,B 0.000,C 90.000,E1 70.369} C_DIS
LIN {X -0.038,Y -308.537,Z 1242.371,A 0.000,B 0.000,C 90.000,E1 66.847} C_DIS
LIN {X 0.101,Y -293.561,Z 1242.351,A 0.000,B 0.000,C 90.000,E1 63.204} C_DIS
LIN {X -0.089,Y -281.218,Z 1242.333,A 0.000,B 0.000,C 90.000,E1 59.871} C_DIS
LIN {X -0.072,Y -269.835,Z 1242.313,A 0.000,B 0.000,C 90.000,E1 56.421} C_DIS
LIN {X 0.007,Y -259.463,Z 1242.294,A 0.000,B 0.000,C 90.000,E1 52.889} C_DIS
LIN {X 0.037,Y -250.048,Z 1242.274,A 0.000,B 0.000,C 90.000,E1 49.299} C_DIS
LIN {X 0.041,Y -241.249,Z 1242.254,A 0.000,B 0.000,C 90.000,E1 45.648} C_DIS
LIN {X -0.096,Y -236.179,Z 1242.241,A 0.000,B 0.000,C 90.000,E1 43.461} C_DIS
LIN {X -0.013,Y -227.964,Z 1242.220,A 0.000,B 0.000,C 90.000,E1 39.688} C_DIS
LIN {X -0.056,Y -220.316,Z 1242.199,A 0.000,B 0.000,C 90.000,E1 35.884} C_DIS
LIN {X -0.045,Y -213.382,Z 1242.178,A 0.000,B 0.000,C 90.000,E1 32.005} C_DIS
LIN {X 0.031,Y -207.384,Z 1242.156,A 0.000,B 0.000,C 90.000,E1 28.052} C_DIS
LIN {X -0.001,Y -202.209,Z 1242.134,A 0.000,B 0.000,C 90.000,E1 24.079} C_DIS
LIN {X -0.046,Y -197.933,Z 1242.111,A 0.000,B 0.000,C 90.000,E1 20.066} C_DIS
LIN {X -0.054,Y -193.851,Z 1242.084,A 0.000,B 0.000,C 90.000,E1 15.190} C_DIS
LIN {X -0.041,Y -190.753,Z 1242.052,A 0.000,B 0.000,C 90.000,E1 9.443} C_DIS
LIN {X -0.098,Y -191.431,Z 1241.970,A 0.000,B 0.000,C 90.000,E1 354.609} C_DIS
LIN {X 0.053,Y -194.846,Z 1241.938,A 0.000,B 0.000,C 90.000,E1 348.814} C_DIS
LIN {X 0.064,Y -198.934,Z 1241.911,A 0.000,B 0.000,C 90.000,E1 343.921} C_DIS
LIN {X 0.069,Y -203.230,Z 1241.888,A 0.000,B 0.000,C 90.000,E1 339.880} C_DIS
LIN {X -0.080,Y -208.238,Z 1241.866,A 0.000,B 0.000,C 90.000,E1 335.921} C_DIS
LIN {X -0.017,Y -213.882,Z 1241.844,A 0.000,B 0.000,C 90.000,E1 331.948} C_DIS
LIN {X -0.030,Y -220.127,Z 1241.822,A 0.000,B 0.000,C 90.000,E1 328.043} C_DIS
LIN {X -0.060,Y -227.069,Z 1241.801,A 0.000,B 0.000,C 90.000,E1 324.196} C_DIS
LIN {X 0.107,Y -234.727,Z 1241.780,A 0.000,B 0.000,C 90.000,E1 320.356} C_DIS
LIN {X 0.100,Y -243.311,Z 1241.759,A 0.000,B 0.000,C 90.000,E1 316.620} C_DIS
LIN {X -0.003,Y -252.101,Z 1241.741,A 0.000,B 0.000,C 90.000,E1 313.338} C_DIS
LIN {X -0.069,Y -259.838,Z 1241.727,A 0.000,B 0.000,C 90.000,E1 310.825} C_DIS
LIN {X 0.027,Y -267.504,Z 1241.715,A 0.000,B 0.000,C 90.000,E1 308.669} C_DIS
LIN {X 0.037,Y -277.659,Z 1241.701,A 0.000,B 0.000,C 90.000,E1 306.217} C_DIS
LIN {X -0.058,Y -288.974,Z 1241.688,A 0.000,B 0.000,C 90.000,E1 303.833} C_DIS
LIN {X 0.019,Y -299.733,Z 1241.677,A 0.000,B 0.000,C 90.000,E1 301.799} C_DIS
LIN {X 0.085,Y -307.616,Z 1241.669,A 0.000,B 0.000,C 90.000,E1 300.463} C_DIS
LIN {X 0.099,Y -316.352,Z 1241.662,A 0.000,B 0.000,C 90.000,E1 299.155} C_DIS
LIN {X -0.025,Y -330.964,Z 1241.651,A 0.000,B 0.000,C 90.000,E1 297.257} C_DIS
LIN {X 0.045,Y -351.737,Z 1241.638,A 0.000,B 0.000,C 90.000,E1 294.771} C_DIS
LIN {X -0.023,Y -370.256,Z 1241.626,A 0.000,B 0.000,C 90.000,E1 292.717} C_DIS
LIN {X 0.067,Y -383.245,Z 1241.618,A 0.000,B 0.000,C 90.000,E1 291.280} C_DIS
LIN {X -0.157,Y -398.691,Z 1241.609,A 0.000,B 0.000,C 90.000,E1 289.631} C_DIS
LIN {X 0.133,Y -411.647,Z 1241.601,A 0.000,B 0.000,C 90.000,E1 288.236} C_DIS
LIN {X 0.126,Y -421.733,Z 1241.595,A 0.000,B 0.000,C 90.000,E1 287.166} C_DIS
LIN {X -0.023,Y -428.843,Z 1241.591,A 0.000,B 0.000,C 90.000,E1 286.386} C_DIS
LIN {X -0.227,Y -435.546,Z 1241.587,A 0.000,B 0.000,C 90.000,E1 285.607} C_DIS
LIN {X 0.039,Y -441.642,Z 1241.582,A 0.000,B 0.000,C 90.000,E1 284.773} C_DIS
LIN {X -0.171,Y -447.144,Z 1241.578,A 0.000,B 0.000,C 90.000,E1 284.008} C_DIS
LIN {X 0.205,Y -451.973,Z 1241.573,A 0.000,B 0.000,C 90.000,E1 283.175} C_DIS
LIN {X 0.085,Y -456.040,Z 1241.569,A 0.000,B 0.000,C 90.000,E1 282.411} C_DIS
LIN {X -0.099,Y -459.412,Z 1241.565,A 0.000,B 0.000,C 90.000,E1 281.658} C_DIS
LIN {X 0.011,Y -461.328,Z 1241.562,A 0.000,B 0.000,C 90.000,E1 281.130} C_DIS
LIN {X 0.125,Y -463.028,Z 1241.559,A 0.000,B 0.000,C 90.000,E1 280.602} C_DIS
LIN {X 0.167,Y -464.473,Z 1241.556,A 0.000,B 0.000,C 90.000,E1 280.084} C_DIS
LIN {X -0.157,Y -465.665,Z 1241.553,A 0.000,B 0.000,C 90.000,E1 279.613} C_DIS
LIN {X -0.092,Y -466.549,Z 1241.550,A 0.000,B 0.000,C 90.000,E1 279.095} C_DIS
LIN {X 0.053,Y -467.160,Z 1241.548,A 0.000,B 0.000,C 90.000,E1 278.568} C_DIS
LIN {X 0.133,Y -467.484,Z 1241.545,A 0.000,B 0.000,C 90.000,E1 278.049} C_DIS
LIN {X -0.246,Y -467.420,Z 1241.542,A 0.000,B 0.000,C 90.000,E1 277.587} C_DIS
LIN {X -0.157,Y -466.940,Z 1241.539,A 0.000,B 0.000,C 90.000,E1 277.068} C_DIS
LIN {X -0.068,Y -466.022,Z 1241.536,A 0.000,B 0.000,C 90.000,E1 276.549} C_DIS
LIN {X 0.018,Y -464.638,Z 1241.534,A 0.000,B 0.000,C 90.000,E1 276.030} C_DIS
LIN {X 0.098,Y -462.862,Z 1241.531,A 0.000,B 0.000,C 90.000,E1 275.511} C_DIS
LIN {X -0.016,Y -459.424,Z 1241.526,A 0.000,B 0.000,C 90.000,E1 274.759} C_DIS
LIN {X -0.008,Y -456.451,Z 1241.524,A 0.000,B 0.000,C 90.000,E1 274.245} C_DIS
LIN {X 0.019,Y -452.802,Z 1241.521,A 0.000,B 0.000,C 90.000,E1 273.726} C_DIS
LIN {X -0.210,Y -450.643,Z 1241.519,A 0.000,B 0.000,C 90.000,E1 273.498} C_DIS
LIN {X -0.214,Y -445.412,Z 1241.516,A 0.000,B 0.000,C 90.000,E1 272.980} C_DIS
LIN {X 0.026,Y -439.275,Z 1241.514,A 0.000,B 0.000,C 90.000,E1 272.465} C_DIS
LIN {X -0.102,Y -432.461,Z 1241.511,A 0.000,B 0.000,C 90.000,E1 272.064} C_DIS
LIN {X -0.074,Y -425.472,Z 1241.510,A 0.000,B 0.000,C 90.000,E1 271.718} C_DIS
LIN {X -0.037,Y -418.356,Z 1241.508,A 0.000,B 0.000,C 90.000,E1 271.432} C_DIS
LIN {X -0.003,Y -411.754,Z 1241.507,A 0.000,B 0.000,C 90.000,E1 271.203} C_DIS
LIN {X -0.192,Y -404.591,Z 1241.506,A 0.000,B 0.000,C 90.000,E1 271.031} C_DIS
LIN {X 0.173,Y -393.935,Z 1241.504,A 0.000,B 0.000,C 90.000,E1 270.745} C_DIS
LIN {X 0.099,Y -381.883,Z 1241.503,A 0.000,B 0.000,C 90.000,E1 270.573} C_DIS
LIN {X 0.007,Y -374.656,Z 1241.503,A 0.000,B 0.000,C 90.000,E1 270.516} C_DIS
LIN {X 0.119,Y -365.042,Z 1241.503,A 0.000,B 0.000,C 90.000,E1 270.458} C_DIS
LIN {X 0.033,Y -181.569,Z 1241.503,A 0.000,B 0.000,C 90.000,E1 270.458} C_DIS
LIN {X -0.052,Y -180.998,Z 1241.484,A 0.000,B 0.000,C 90.000,E1 267.078} C_DIS
LIN {X 0.065,Y -180.906,Z 1241.474,A 0.000,B 0.000,C 90.000,E1 265.355} C_DIS
LIN {X -0.041,Y -180.692,Z 1241.470,A 0.000,B 0.000,C 90.000,E1 264.546} C_DIS
LIN {X 0.036,Y -178.776,Z 1241.442,A 0.000,B 0.000,C 90.000,E1 259.454} C_DIS
LIN {X -0.061,Y -175.823,Z 1241.413,A 0.000,B 0.000,C 90.000,E1 254.393} C_DIS
LIN {X -0.060,Y -172.010,Z 1241.385,A 0.000,B 0.000,C 90.000,E1 249.263} C_DIS
LIN {X -0.084,Y -171.430,Z 1241.380,A 0.000,B 0.000,C 90.000,E1 248.411} C_DIS
LIN {X -0.028,Y -167.666,Z 1241.356,A 0.000,B 0.000,C 90.000,E1 244.076} C_DIS
LIN {X -0.088,Y -166.338,Z 1241.346,A 0.000,B 0.000,C 90.000,E1 242.359} C_DIS
LIN {X -0.095,Y -163.075,Z 1241.327,A 0.000,B 0.000,C 90.000,E1 238.869} C_DIS
LIN {X -0.043,Y -161.015,Z 1241.312,A 0.000,B 0.000,C 90.000,E1 236.215} C_DIS
LIN {X 0.066,Y -157.758,Z 1241.293,A 0.000,B 0.000,C 90.000,E1 232.637} C_DIS
LIN {X 0.004,Y -155.796,Z 1241.278,A 0.000,B 0.000,C 90.000,E1 229.989} C_DIS
LIN {X 0.059,Y -152.048,Z 1241.253,A 0.000,B 0.000,C 90.000,E1 225.486} C_DIS
LIN {X 0.076,Y -150.297,Z 1241.238,A 0.000,B 0.000,C 90.000,E1 222.771} C_DIS
LIN {X 0.002,Y -147.044,Z 1241.213,A 0.000,B 0.000,C 90.000,E1 218.257} C_DIS
LIN {X -0.006,Y -145.624,Z 1241.197,A 0.000,B 0.000,C 90.000,E1 215.518} C_DIS
LIN {X -0.008,Y -143.007,Z 1241.172,A 0.000,B 0.000,C 90.000,E1 210.924} C_DIS
LIN {X -0.076,Y -141.634,Z 1241.151,A 0.000,B 0.000,C 90.000,E1 207.257} C_DIS
LIN {X -0.025,Y -139.437,Z 1241.115,A 0.000,B 0.000,C 90.000,E1 200.737} C_DIS
LIN {X 0.029,Y -139.169,Z 1241.105,A 0.000,B 0.000,C 90.000,E1 198.852} C_DIS
LIN {X 0.062,Y -138.317,Z 1241.053,A 0.000,B 0.000,C 90.000,E1 189.500} C_DIS
LIN {X -0.065,Y -139.475,Z 1241.006,A 0.000,B 0.000,C 90.000,E1 181.146} C_DIS
LIN {X 0.016,Y -141.052,Z 1240.975,A 0.000,B 0.000,C 90.000,E1 175.527} C_DIS
LIN {X -0.031,Y -142.424,Z 1240.960,A 0.000,B 0.000,C 90.000,E1 172.761} C_DIS
LIN {X 0.030,Y -144.660,Z 1240.934,A 0.000,B 0.000,C 90.000,E1 168.117} C_DIS
LIN {X 0.015,Y -147.243,Z 1240.914,A 0.000,B 0.000,C 90.000,E1 164.448} C_DIS
LIN {X 0.032,Y -150.560,Z 1240.888,A 0.000,B 0.000,C 90.000,E1 159.880} C_DIS
LIN {X -0.029,Y -154.027,Z 1240.868,A 0.000,B 0.000,C 90.000,E1 156.282} C_DIS
LIN {X 0.040,Y -157.443,Z 1240.848,A 0.000,B 0.000,C 90.000,E1 152.666} C_DIS
LIN {X -0.011,Y -161.660,Z 1240.828,A 0.000,B 0.000,C 90.000,E1 149.125} C_DIS
LIN {X 0.006,Y -165.855,Z 1240.809,A 0.000,B 0.000,C 90.000,E1 145.595} C_DIS
LIN {X -0.002,Y -170.830,Z 1240.790,A 0.000,B 0.000,C 90.000,E1 142.110} C_DIS
LIN {X 0.046,Y -175.700,Z 1240.770,A 0.000,B 0.000,C 90.000,E1 138.647} C_DIS
LIN {X 0.037,Y -181.312,Z 1240.751,A 0.000,B 0.000,C 90.000,E1 135.243} C_DIS
LIN {X -0.092,Y -186.796,Z 1240.733,A 0.000,B 0.000,C 90.000,E1 131.919} C_DIS
LIN {X -0.021,Y -191.386,Z 1240.719,A 0.000,B 0.000,C 90.000,E1 129.402} C_DIS
LIN {X 0.061,Y -197.230,Z 1240.701,A 0.000,B 0.000,C 90.000,E1 126.091} C_DIS
LIN {X -0.033,Y -200.670,Z 1240.691,A 0.000,B 0.000,C 90.000,E1 124.405} C_DIS
LIN {X -0.086,Y -310.102,Z 1240.691,A 0.000,B 0.000,C 90.000,E1 124.405} C_DIS
LIN {X 0.142,Y -312.476,Z 1240.691,A 0.000,B 0.000,C 90.000,E1 124.326} C_DIS
LIN {X -0.095,Y -316.269,Z 1240.690,A 0.000,B 0.000,C 90.000,E1 124.199} C_DIS
LIN {X 0.107,Y -318.508,Z 1240.689,A 0.000,B 0.000,C 90.000,E1 123.992} C_DIS
LIN {X 0.072,Y -321.608,Z 1240.687,A 0.000,B 0.000,C 90.000,E1 123.658} C_DIS
LIN {X -0.003,Y -323.575,Z 1240.685,A 0.000,B 0.000,C 90.000,E1 123.372} C_DIS
LIN {X -0.080,Y -325.111,Z 1240.684,A 0.000,B 0.000,C 90.000,E1 123.086} C_DIS
LIN {X -0.065,Y -328.654,Z 1240.678,A 0.000,B 0.000,C 90.000,E1 122.133} C_DIS
LIN {X 0.127,Y -339.610,Z 1240.663,A 0.000,B 0.000,C 90.000,E1 119.283} C_DIS
LIN {X 0.010,Y -351.946,Z 1240.647,A 0.000,B 0.000,C 90.000,E1 116.539} C_DIS
LIN {X 0.076,Y -365.778,Z 1240.632,A 0.000,B 0.000,C 90.000,E1 113.823} C_DIS
LIN {X 0.135,Y -379.420,Z 1240.619,A 0.000,B 0.000,C 90.000,E1 111.461} C_DIS
LIN {X -0.238,Y -394.432,Z 1240.607,A 0.000,B 0.000,C 90.000,E1 109.214} C_DIS
LIN {X 0.136,Y -410.918,Z 1240.594,A 0.000,B 0.000,C 90.000,E1 106.913} C_DIS
LIN {X 0.179,Y -428.996,Z 1240.582,A 0.000,B 0.000,C 90.000,E1 104.717} C_DIS
LIN {X -0.144,Y -448.606,Z 1240.570,A 0.000,B 0.000,C 90.000,E1 102.647} C_DIS
LIN {X 0.167,Y -468.905,Z 1240.559,A 0.000,B 0.000,C 90.000,E1 100.658} C_DIS
LIN {X 0.160,Y -473.961,Z 1240.557,A 0.000,B 0.000,C 90.000,E1 100.197} C_DIS
LIN {X 0.163,Y -475.924,Z 1240.555,A 0.000,B 0.000,C 90.000,E1 99.962} C_DIS
LIN {X 0.165,Y -477.418,Z 1240.554,A 0.000,B 0.000,C 90.000,E1 99.726} C_DIS
LIN {X -0.045,Y -478.626,Z 1240.553,A 0.000,B 0.000,C 90.000,E1 99.500} C_DIS
LIN {X -0.175,Y -479.506,Z 1240.551,A 0.000,B 0.000,C 90.000,E1 99.265} C_DIS
LIN {X -0.025,Y -480.441,Z 1240.549,A 0.000,B 0.000,C 90.000,E1 98.746} C_DIS
LIN {X 0.202,Y -480.388,Z 1240.546,A 0.000,B 0.000,C 90.000,E1 98.219} C_DIS
LIN {X -0.111,Y -479.344,Z 1240.543,A 0.000,B 0.000,C 90.000,E1 97.757} C_DIS
LIN {X 0.177,Y -478.403,Z 1240.542,A 0.000,B 0.000,C 90.000,E1 97.473} C_DIS
LIN {X 0.053,Y -477.124,Z 1240.540,A 0.000,B 0.000,C 90.000,E1 97.239} C_DIS
LIN {X 0.204,Y -473.500,Z 1240.537,A 0.000,B 0.000,C 90.000,E1 96.720} C_DIS
LIN {X -0.057,Y -453.609,Z 1240.522,A 0.000,B 0.000,C 90.000,E1 93.955} C_DIS
LIN {X -0.111,Y -434.858,Z 1240.506,A 0.000,B 0.000,C 90.000,E1 91.088} C_DIS
LIN {X -0.129,Y -420.942,Z 1240.493,A 0.000,B 0.000,C 90.000,E1 88.682} C_DIS
LIN {X 0.034,Y -406.594,Z 1240.477,A 0.000,B 0.000,C 90.000,E1 85.927} C_DIS
LIN {X 0.090,Y -396.452,Z 1240.467,A 0.000,B 0.000,C 90.000,E1 83.970} C_DIS
LIN {X -0.029,Y -386.229,Z 1240.456,A 0.000,B 0.000,C 90.000,E1 82.008} C_DIS
LIN {X 0.049,Y -377.292,Z 1240.446,A 0.000,B 0.000,C 90.000,E1 80.274} C_DIS
LIN {X 0.095,Y -369.637,Z 1240.438,A 0.000,B 0.000,C 90.000,E1 78.814} C_DIS
LIN {X -0.005,Y -360.187,Z 1240.428,A 0.000,B 0.000,C 90.000,E1 77.061} C_DIS
LIN {X -0.109,Y -350.477,Z 1240.418,A 0.000,B 0.000,C 90.000,E1 75.283} C_DIS
LIN {X -0.050,Y -339.074,Z 1240.406,A 0.000,B 0.000,C 90.000,E1 73.142} C_DIS
LIN {X -0.065,Y -326.415,Z 1240.392,A 0.000,B 0.000,C 90.000,E1 70.659} C_DIS
LIN {X -0.077,Y -309.769,Z 1240.373,A 0.000,B 0.000,C 90.000,E1 67.155} C_DIS
LIN {X 0.105,Y -294.673,Z 1240.353,A 0.000,B 0.000,C 90.000,E1 63.512} C_DIS
LIN {X -0.043,Y -282.197,Z 1240.334,A 0.000,B 0.000,C 90.000,E1 60.177} C_DIS
LIN {X 0.093,Y -270.688,Z 1240.315,A 0.000,B 0.000,C 90.000,E1 56.707} C_DIS
LIN {X -0.025,Y -261.198,Z 1240.298,A 0.000,B 0.000,C 90.000,E1 53.577} C_DIS
LIN {X 0.047,Y -251.573,Z 1240.278,A 0.000,B 0.000,C 90.000,E1 49.989} C_DIS
LIN {X -0.070,Y -242.622,Z 1240.258,A 0.000,B 0.000,C 90.000,E1 46.377} C_DIS
LIN {X 0.097,Y -235.811,Z 1240.241,A 0.000,B 0.000,C 90.000,E1 43.380} C_DIS
LIN {X 0.014,Y -227.553,Z 1240.220,A 0.000,B 0.000,C 90.000,E1 39.644} C_DIS
LIN {X 0.094,Y -219.868,Z 1240.199,A 0.000,B 0.000,C 90.000,E1 35.804} C_DIS
LIN {X 0.084,Y -212.936,Z 1240.177,A 0.000,B 0.000,C 90.000,E1 31.926} C_DIS
LIN {X -0.045,Y -206.950,Z 1240.156,A 0.000,B 0.000,C 90.000,E1 28.025} C_DIS
LIN {X 0.001,Y -201.758,Z 1240.133,A 0.000,B 0.000,C 90.000,E1 24.027} C_DIS
LIN {X 0.015,Y -197.510,Z 1240.111,A 0.000,B 0.000,C 90.000,E1 19.993} C_DIS
LIN {X -0.070,Y -193.473,Z 1240.084,A 0.000,B 0.000,C 90.000,E1 15.134} C_DIS
LIN {X -0.038,Y -190.420,Z 1240.052,A 0.000,B 0.000,C 90.000,E1 9.378} C_DIS
LIN {X 0.081,Y -191.138,Z 1239.970,A 0.000,B 0.000,C 90.000,E1 354.552} C_DIS
LIN {X 0.029,Y -194.575,Z 1239.938,A 0.000,B 0.000,C 90.000,E1 348.814} C_DIS
LIN {X 0.030,Y -198.687,Z 1239.911,A 0.000,B 0.000,C 90.000,E1 343.921} C_DIS
LIN {X 0.028,Y -203.012,Z 1239.888,A 0.000,B 0.000,C 90.000,E1 339.880} C_DIS
LIN {X 0.059,Y -208.047,Z 1239.866,A 0.000,B 0.000,C 90.000,E1 335.869} C_DIS
LIN {X 0.114,Y -213.753,Z 1239.844,A 0.000,B 0.000,C 90.000,E1 331.897} C_DIS
LIN {X 0.094,Y -220.017,Z 1239.822,A 0.000,B 0.000,C 90.000,E1 327.995} C_DIS
LIN {X -0.129,Y -226.951,Z 1239.801,A 0.000,B 0.000,C 90.000,E1 324.196} C_DIS
LIN {X 0.032,Y -234.637,Z 1239.780,A 0.000,B 0.000,C 90.000,E1 320.356} C_DIS
LIN {X 0.021,Y -243.210,Z 1239.759,A 0.000,B 0.000,C 90.000,E1 316.620} C_DIS
LIN {X 0.084,Y -252.033,Z 1239.741,A 0.000,B 0.000,C 90.000,E1 313.299} C_DIS
LIN {X 0.037,Y -259.789,Z 1239.727,A 0.000,B 0.000,C 90.000,E1 310.782} C_DIS
LIN {X 0.082,Y -266.122,Z 1239.717,A 0.000,B 0.000,C 90.000,E1 308.991} C_DIS
LIN {X 0.143,Y -274.629,Z 1239.705,A 0.000,B 0.000,C 90.000,E1 306.870} C_DIS
LIN {X 0.034,Y -283.955,Z 1239.693,A 0.000,B 0.000,C 90.000,E1 304.818} C_DIS
LIN {X -0.069,Y -294.182,Z 1239.682,A 0.000,B 0.000,C 90.000,E1 302.801} C_DIS
LIN {X -0.048,Y -305.473,Z 1239.671,A 0.000,B 0.000,C 90.000,E1 300.797} C_DIS
LIN {X 0.091,Y -313.976,Z 1239.664,A 0.000,B 0.000,C 90.000,E1 299.461} C_DIS
LIN {X 0.112,Y -325.825,Z 1239.655,A 0.000,B 0.000,C 90.000,E1 297.847} C_DIS
LIN {X 0.034,Y -348.830,Z 1239.639,A 0.000,B 0.000,C 90.000,E1 295.079} C_DIS
LIN {X -0.021,Y -367.346,Z 1239.628,A 0.000,B 0.000,C 90.000,E1 293.003} C_DIS
LIN {X 0.132,Y -377.844,Z 1239.621,A 0.000,B 0.000,C 90.000,E1 291.844} C_DIS
LIN {X 0.172,Y -390.783,Z 1239.614,A 0.000,B 0.000,C 90.000,E1 290.429} C_DIS
LIN {X 0.020,Y -408.756,Z 1239.603,A 0.000,B 0.000,C 90.000,E1 288.544} C_DIS
LIN {X 0.202,Y -418.881,Z 1239.597,A 0.000,B 0.000,C 90.000,E1 287.457} C_DIS
LIN {X 0.067,Y -426.158,Z 1239.593,A 0.000,B 0.000,C 90.000,E1 286.677} C_DIS
LIN {X -0.131,Y -433.014,Z 1239.588,A 0.000,B 0.000,C 90.000,E1 285.898} C_DIS
LIN {X 0.118,Y -439.333,Z 1239.584,A 0.000,B 0.000,C 90.000,E1 285.064} C_DIS
LIN {X -0.120,Y -445.104,Z 1239.579,A 0.000,B 0.000,C 90.000,E1 284.300} C_DIS
LIN {X 0.137,Y -450.186,Z 1239.575,A 0.000,B 0.000,C 90.000,E1 283.480} C_DIS
LIN {X 0.000,Y -454.554,Z 1239.571,A 0.000,B 0.000,C 90.000,E1 282.715} C_DIS
LIN {X -0.094,Y -458.191,Z 1239.566,A 0.000,B 0.000,C 90.000,E1 281.951} C_DIS
LIN {X -0.165,Y -461.224,Z 1239.562,A 0.000,B 0.000,C 90.000,E1 281.186} C_DIS
LIN {X -0.053,Y -462.930,Z 1239.559,A 0.000,B 0.000,C 90.000,E1 280.658} C_DIS
LIN {X -0.013,Y -464.398,Z 1239.556,A 0.000,B 0.000,C 90.000,E1 280.141} C_DIS
LIN {X 0.122,Y -465.606,Z 1239.553,A 0.000,B 0.000,C 90.000,E1 279.613} C_DIS
LIN {X 0.186,Y -466.540,Z 1239.551,A 0.000,B 0.000,C 90.000,E1 279.095} C_DIS
LIN {X -0.130,Y -467.190,Z 1239.548,A 0.000,B 0.000,C 90.000,E1 278.624} C_DIS
LIN {X -0.052,Y -467.545,Z 1239.545,A 0.000,B 0.000,C 90.000,E1 278.106} C_DIS
LIN {X 0.033,Y -467.506,Z 1239.542,A 0.000,B 0.000,C 90.000,E1 277.587} C_DIS
LIN {X 0.121,Y -467.084,Z 1239.539,A 0.000,B 0.000,C 90.000,E1 277.068} C_DIS
LIN {X -0.253,Y -466.220,Z 1239.536,A 0.000,B 0.000,C 90.000,E1 276.606} C_DIS
LIN {X -0.166,Y -464.921,Z 1239.534,A 0.000,B 0.000,C 90.000,E1 276.087} C_DIS
LIN {X -0.084,Y -463.208,Z 1239.531,A 0.000,B 0.000,C 90.000,E1 275.568} C_DIS
LIN {X -0.012,Y -461.063,Z 1239.528,A 0.000,B 0.000,C 90.000,E1 275.049} C_DIS
LIN {X 0.048,Y -458.469,Z 1239.525,A 0.000,B 0.000,C 90.000,E1 274.531} C_DIS
LIN {X 0.085,Y -455.281,Z 1239.522,A 0.000,B 0.000,C 90.000,E1 274.012} C_DIS
LIN {X 0.076,Y -451.225,Z 1239.520,A 0.000,B 0.000,C 90.000,E1 273.498} C_DIS
LIN {X -0.162,Y -448.835,Z 1239.518,A 0.000,B 0.000,C 90.000,E1 273.269} C_DIS
LIN {X -0.048,Y -443.253,Z 1239.515,A 0.000,B 0.000,C 90.000,E1 272.751} C_DIS
LIN {X -0.166,Y -440.060,Z 1239.514,A 0.000,B 0.000,C 90.000,E1 272.522} C_DIS
LIN {X 0.111,Y -433.393,Z 1239.512,A 0.000,B 0.000,C 90.000,E1 272.064} C_DIS
LIN {X 0.074,Y -426.376,Z 1239.510,A 0.000,B 0.000,C 90.000,E1 271.718} C_DIS
LIN {X 0.080,Y -419.358,Z 1239.508,A 0.000,B 0.000,C 90.000,E1 271.432} C_DIS
LIN {X 0.032,Y -412.517,Z 1239.507,A 0.000,B 0.000,C 90.000,E1 271.203} C_DIS
LIN {X -0.178,Y -405.426,Z 1239.506,A 0.000,B 0.000,C 90.000,E1 271.031} C_DIS
LIN {X 0.128,Y -394.430,Z 1239.504,A 0.000,B 0.000,C 90.000,E1 270.745} C_DIS
LIN {X 0.013,Y -386.584,Z 1239.504,A 0.000,B 0.000,C 90.000,E1 270.630} C_DIS
LIN {X -0.100,Y -374.837,Z 1239.503,A 0.000,B 0.000,C 90.000,E1 270.516} C_DIS
LIN {X 0.012,Y -365.964,Z 1239.503,A 0.000,B 0.000,C 90.000,E1 270.458} C_DIS
LIN {X -0.020,Y -181.571,Z 1239.503,A 0.000,B 0.000,C 90.000,E1 270.458} C_DIS
LIN {X 0.014,Y -180.906,Z 1239.474,A 0.000,B 0.000,C 90.000,E1 265.355} C_DIS
LIN {X 0.088,Y -180.684,Z 1239.469,A 0.000,B 0.000,C 90.000,E1 264.489} C_DIS
LIN {X -0.014,Y -178.767,Z 1239.441,A 0.000,B 0.000,C 90.000,E1 259.454} C_DIS
LIN {X 0.058,Y -175.814,Z 1239.413,A 0.000,B 0.000,C 90.000,E1 254.338} C_DIS
LIN {X 0.052,Y -172.001,Z 1239.385,A 0.000,B 0.000,C 90.000,E1 249.209} C_DIS
LIN {X 0.026,Y -171.415,Z 1239.380,A 0.000,B 0.000,C 90.000,E1 248.358} C_DIS
LIN {X 0.073,Y -167.654,Z 1239.356,A 0.000,B 0.000,C 90.000,E1 244.024} C_DIS
LIN {X 0.088,Y -166.320,Z 1239.346,A 0.000,B 0.000,C 90.000,E1 242.281} C_DIS
LIN {X -0.003,Y -163.062,Z 1239.327,A 0.000,B 0.000,C 90.000,E1 238.820} C_DIS
LIN {X 0.043,Y -160.998,Z 1239.312,A 0.000,B 0.000,C 90.000,E1 236.167} C_DIS
LIN {X 0.019,Y -157.745,Z 1239.292,A 0.000,B 0.000,C 90.000,E1 232.637} C_DIS
LIN {X -0.042,Y -155.782,Z 1239.278,A 0.000,B 0.000,C 90.000,E1 229.989} C_DIS
LIN {X 0.012,Y -152.036,Z 1239.253,A 0.000,B 0.000,C 90.000,E1 225.486} C_DIS
LIN {X 0.030,Y -150.285,Z 1239.238,A 0.000,B 0.000,C 90.000,E1 222.771} C_DIS
LIN {X -0.043,Y -147.034,Z 1239.212,A 0.000,B 0.000,C 90.000,E1 218.257} C_DIS
LIN {X -0.051,Y -145.614,Z 1239.197,A 0.000,B 0.000,C 90.000,E1 215.518} C_DIS
LIN {X -0.052,Y -142.999,Z 1239.172,A 0.000,B 0.000,C 90.000,E1 210.924} C_DIS
LIN {X 0.007,Y -141.626,Z 1239.151,A 0.000,B 0.000,C 90.000,E1 207.206} C_DIS
LIN {X -0.068,Y -139.433,Z 1239.115,A 0.000,B 0.000,C 90.000,E1 200.737} C_DIS
LIN {X -0.014,Y -139.165,Z 1239.105,A 0.000,B 0.000,C 90.000,E1 198.852} C_DIS
LIN {X 0.023,Y -138.340,Z 1239.058,A 0.000,B 0.000,C 90.000,E1 190.433} C_DIS
LIN {X 0.030,Y -139.477,Z 1239.006,A 0.000,B 0.000,C 90.000,E1 181.088} C_DIS
LIN {X -0.029,Y -141.060,Z 1238.975,A 0.000,B 0.000,C 90.000,E1 175.527} C_DIS
LIN {X 0.066,Y -142.433,Z 1238.960,A 0.000,B 0.000,C 90.000,E1 172.704} C_DIS
LIN {X -0.014,Y -144.671,Z 1238.934,A 0.000,B 0.000,C 90.000,E1 168.117} C_DIS
LIN {X -0.031,Y -147.257,Z 1238.914,A 0.000,B 0.000,C 90.000,E1 164.448} C_DIS
LIN {X -0.014,Y -150.575,Z 1238.888,A 0.000,B 0.000,C 90.000,E1 159.880} C_DIS
LIN {X 0.066,Y -154.044,Z 1238.868,A 0.000,B 0.000,C 90.000,E1 156.230} C_DIS
LIN {X -0.007,Y -157.462,Z 1238.848,A 0.000,B 0.000,C 90.000,E1 152.666} C_DIS
LIN {X -0.059,Y -161.682,Z 1238.828,A 0.000,B 0.000,C 90.000,E1 149.125} C_DIS
LIN {X -0.042,Y -165.877,Z 1238.809,A 0.000,B 0.000,C 90.000,E1 145.595} C_DIS
LIN {X -0.052,Y -170.856,Z 1238.789,A 0.000,B 0.000,C 90.000,E1 142.110} C_DIS
LIN {X -0.006,Y -175.725,Z 1238.770,A 0.000,B 0.000,C 90.000,E1 138.647} C_DIS
LIN {X -0.014,Y -181.336,Z 1238.751,A 0.000,B 0.000,C 90.000,E1 135.243} C_DIS
LIN {X -0.019,Y -186.824,Z 1238.733,A 0.000,B 0.000,C 90.000,E1 131.881} C_DIS
LIN {X 0.074,Y -191.412,Z 1238.719,A 0.000,B 0.000,C 90.000,E1 129.358} C_DIS
LIN {X 0.008,Y -197.260,Z 1238.701,A 0.000,B 0.000,C 90.000,E1 126.091} C_DIS
LIN {X 0.023,Y -200.728,Z 1238.691,A 0.000,B 0.000,C 90.000,E1 124.358} C_DIS
LIN {X 0.159,Y -310.984,Z 1238.691,A 0.000,B 0.000,C 90.000,E1 124.326} C_DIS
LIN {X 0.058,Y -312.069,Z 1238.691,A 0.000,B 0.000,C 90.000,E1 124.326} C_DIS
LIN {X -0.180,Y -316.155,Z 1238.690,A 0.000,B 0.000,C 90.000,E1 124.199} C_DIS
LIN {X 0.021,Y -318.449,Z 1238.689,A 0.000,B 0.000,C 90.000,E1 123.992} C_DIS
LIN {X -0.015,Y -321.593,Z 1238.687,A 0.000,B 0.000,C 90.000,E1 123.658} C_DIS
LIN {X -0.073,Y -323.563,Z 1238.685,A 0.000,B 0.000,C 90.000,E1 123.372} C_DIS
LIN {X -0.132,Y -325.104,Z 1238.684,A 0.000,B 0.000,C 90.000,E1 123.086} C_DIS
LIN {X 0.056,Y -327.530,Z 1238.680,A 0.000,B 0.000,C 90.000,E1 122.418} C_DIS
LIN {X -0.065,Y -338.340,Z 1238.664,A 0.000,B 0.000,C 90.000,E1 119.617} C_DIS
LIN {X 0.089,Y -350.525,Z 1238.649,A 0.000,B 0.000,C 90.000,E1 116.821} C_DIS
LIN {X -0.046,Y -364.187,Z 1238.634,A 0.000,B 0.000,C 90.000,E1 114.131} C_DIS
LIN {X -0.034,Y -377.669,Z 1238.621,A 0.000,B 0.000,C 90.000,E1 111.770} C_DIS
LIN {X 0.045,Y -392.509,Z 1238.608,A 0.000,B 0.000,C 90.000,E1 109.450} C_DIS
LIN {X -0.134,Y -408.810,Z 1238.596,A 0.000,B 0.000,C 90.000,E1 107.221} C_DIS
LIN {X -0.037,Y -426.688,Z 1238.583,A 0.000,B 0.000,C 90.000,E1 105.009} C_DIS
LIN {X -0.044,Y -446.146,Z 1238.572,A 0.000,B 0.000,C 90.000,E1 102.883} C_DIS
LIN {X 0.106,Y -466.377,Z 1238.561,A 0.000,B 0.000,C 90.000,E1 100.894} C_DIS
LIN {X 0.100,Y -473.986,Z 1238.557,A 0.000,B 0.000,C 90.000,E1 100.197} C_DIS
LIN {X 0.088,Y -475.922,Z 1238.555,A 0.000,B 0.000,C 90.000,E1 99.962} C_DIS
LIN {X 0.076,Y -477.394,Z 1238.554,A 0.000,B 0.000,C 90.000,E1 99.726} C_DIS
LIN {X -0.133,Y -478.574,Z 1238.553,A 0.000,B 0.000,C 90.000,E1 99.500} C_DIS
LIN {X 0.209,Y -479.431,Z 1238.551,A 0.000,B 0.000,C 90.000,E1 99.208} C_DIS
LIN {X -0.115,Y -480.325,Z 1238.548,A 0.000,B 0.000,C 90.000,E1 98.746} C_DIS
LIN {X 0.112,Y -480.235,Z 1238.546,A 0.000,B 0.000,C 90.000,E1 98.219} C_DIS
LIN {X -0.201,Y -479.150,Z 1238.543,A 0.000,B 0.000,C 90.000,E1 97.757} C_DIS
LIN {X 0.086,Y -478.184,Z 1238.542,A 0.000,B 0.000,C 90.000,E1 97.473} C_DIS
LIN {X -0.039,Y -476.877,Z 1238.540,A 0.000,B 0.000,C 90.000,E1 97.239} C_DIS
LIN {X 0.089,Y -467.662,Z 1238.533,A 0.000,B 0.000,C 90.000,E1 95.967} C_DIS
LIN {X 0.068,Y -451.597,Z 1238.520,A 0.000,B 0.000,C 90.000,E1 93.669} C_DIS
LIN {X -0.052,Y -432.984,Z 1238.504,A 0.000,B 0.000,C 90.000,E1 90.802} C_DIS
LIN {X 0.005,Y -417.752,Z 1238.490,A 0.000,B 0.000,C 90.000,E1 88.108} C_DIS
LIN {X -0.072,Y -406.355,Z 1238.477,A 0.000,B 0.000,C 90.000,E1 85.927} C_DIS
LIN {X -0.019,Y -396.206,Z 1238.466,A 0.000,B 0.000,C 90.000,E1 83.970} C_DIS
LIN {X -0.141,Y -385.980,Z 1238.455,A 0.000,B 0.000,C 90.000,E1 82.008} C_DIS
LIN {X -0.064,Y -377.048,Z 1238.446,A 0.000,B 0.000,C 90.000,E1 80.274} C_DIS
LIN {X -0.027,Y -367.826,Z 1238.436,A 0.000,B 0.000,C 90.000,E1 78.522} C_DIS
LIN {X -0.075,Y -358.357,Z 1238.426,A 0.000,B 0.000,C 90.000,E1 76.756} C_DIS
LIN {X 0.046,Y -348.634,Z 1238.416,A 0.000,B 0.000,C 90.000,E1 74.936} C_DIS
LIN {X 0.046,Y -335.652,Z 1238.403,A 0.000,B 0.000,C 90.000,E1 72.489} C_DIS
LIN {X -0.060,Y -323.078,Z 1238.389,A 0.000,B 0.000,C 90.000,E1 70.007} C_DIS
LIN {X -0.082,Y -306.726,Z 1238.369,A 0.000,B 0.000,C 90.000,E1 66.485} C_DIS
LIN {X -0.146,Y -291.905,Z 1238.349,A 0.000,B 0.000,C 90.000,E1 62.871} C_DIS
LIN {X 0.013,Y -279.587,Z 1238.330,A 0.000,B 0.000,C 90.000,E1 59.459} C_DIS
LIN {X 0.054,Y -269.357,Z 1238.313,A 0.000,B 0.000,C 90.000,E1 56.342} C_DIS
LIN {X -0.039,Y -258.927,Z 1238.294,A 0.000,B 0.000,C 90.000,E1 52.844} C_DIS
LIN {X -0.034,Y -249.412,Z 1238.274,A 0.000,B 0.000,C 90.000,E1 49.256} C_DIS
LIN {X 0.111,Y -240.583,Z 1238.253,A 0.000,B 0.000,C 90.000,E1 45.567} C_DIS
LIN {X -0.040,Y -235.437,Z 1238.241,A 0.000,B 0.000,C 90.000,E1 43.380} C_DIS
LIN {X -0.129,Y -227.146,Z 1238.220,A 0.000,B 0.000,C 90.000,E1 39.644} C_DIS
LIN {X -0.056,Y -219.421,Z 1238.199,A 0.000,B 0.000,C 90.000,E1 35.804} C_DIS
LIN {X -0.076,Y -212.493,Z 1238.177,A 0.000,B 0.000,C 90.000,E1 31.926} C_DIS
LIN {X -0.031,Y -206.504,Z 1238.155,A 0.000,B 0.000,C 90.000,E1 27.975} C_DIS
LIN {X 0.088,Y -201.314,Z 1238.133,A 0.000,B 0.000,C 90.000,E1 23.951} C_DIS
LIN {X 0.012,Y -197.098,Z 1238.111,A 0.000,B 0.000,C 90.000,E1 19.939} C_DIS
LIN {X -0.032,Y -193.099,Z 1238.084,A 0.000,B 0.000,C 90.000,E1 15.064} C_DIS
LIN {X -0.062,Y -190.082,Z 1238.052,A 0.000,B 0.000,C 90.000,E1 9.321} C_DIS
LIN {X 0.070,Y -190.842,Z 1237.970,A 0.000,B 0.000,C 90.000,E1 354.552} C_DIS
LIN {X 0.006,Y -194.291,Z 1237.938,A 0.000,B 0.000,C 90.000,E1 348.814} C_DIS
LIN {X -0.005,Y -198.433,Z 1237.911,A 0.000,B 0.000,C 90.000,E1 343.921} C_DIS
LIN {X -0.015,Y -202.792,Z 1237.888,A 0.000,B 0.000,C 90.000,E1 339.880} C_DIS
LIN {X 0.009,Y -207.856,Z 1237.866,A 0.000,B 0.000,C 90.000,E1 335.869} C_DIS
LIN {X 0.055,Y -213.620,Z 1237.844,A 0.000,B 0.000,C 90.000,E1 331.897} C_DIS
LIN {X 0.029,Y -219.877,Z 1237.822,A 0.000,B 0.000,C 90.000,E1 327.995} C_DIS
LIN {X 0.067,Y -225.399,Z 1237.805,A 0.000,B 0.000,C 90.000,E1 324.895} C_DIS
LIN {X 0.043,Y -232.905,Z 1237.784,A 0.000,B 0.000,C 90.000,E1 321.090} C_DIS
LIN {X 0.161,Y -241.296,Z 1237.763,A 0.000,B 0.000,C 90.000,E1 317.310} C_DIS
LIN {X 0.001,Y -249.888,Z 1237.745,A 0.000,B 0.000,C 90.000,E1 314.028} C_DIS
LIN {X -0.083,Y -258.558,Z 1237.729,A 0.000,B 0.000,C 90.000,E1 311.148} C_DIS
LIN {X -0.067,Y -264.758,Z 1237.719,A 0.000,B 0.000,C 90.000,E1 309.358} C_DIS
LIN {X -0.036,Y -273.104,Z 1237.707,A 0.000,B 0.000,C 90.000,E1 307.237} C_DIS
LIN {X -0.064,Y -283.900,Z 1237.693,A 0.000,B 0.000,C 90.000,E1 304.818} C_DIS
LIN {X 0.076,Y -294.131,Z 1237.682,A 0.000,B 0.000,C 90.000,E1 302.752} C_DIS
LIN {X -0.155,Y -305.370,Z 1237.671,A 0.000,B 0.000,C 90.000,E1 300.797} C_DIS
LIN {X -0.021,Y -313.844,Z 1237.664,A 0.000,B 0.000,C 90.000,E1 299.461} C_DIS
LIN {X -0.005,Y -325.713,Z 1237.655,A 0.000,B 0.000,C 90.000,E1 297.847} C_DIS
LIN {X 0.010,Y -348.583,Z 1237.639,A 0.000,B 0.000,C 90.000,E1 295.079} C_DIS
LIN {X -0.100,Y -366.995,Z 1237.628,A 0.000,B 0.000,C 90.000,E1 293.025} C_DIS
LIN {X -0.149,Y -377.549,Z 1237.622,A 0.000,B 0.000,C 90.000,E1 291.897} C_DIS
LIN {X 0.091,Y -393.165,Z 1237.612,A 0.000,B 0.000,C 90.000,E1 290.174} C_DIS
LIN {X -0.041,Y -411.015,Z 1237.602,A 0.000,B 0.000,C 90.000,E1 288.308} C_DIS
LIN {X 0.141,Y -421.074,Z 1237.596,A 0.000,B 0.000,C 90.000,E1 287.221} C_DIS
LIN {X -0.092,Y -428.328,Z 1237.591,A 0.000,B 0.000,C 90.000,E1 286.441} C_DIS
LIN {X 0.116,Y -435.088,Z 1237.587,A 0.000,B 0.000,C 90.000,E1 285.607} C_DIS
LIN {X -0.043,Y -441.226,Z 1237.582,A 0.000,B 0.000,C 90.000,E1 284.828} C_DIS
LIN {X 0.174,Y -446.762,Z 1237.578,A 0.000,B 0.000,C 90.000,E1 284.008} C_DIS
LIN {X 0.008,Y -451.654,Z 1237.574,A 0.000,B 0.000,C 90.000,E1 283.244} C_DIS
LIN {X -0.113,Y -455.786,Z 1237.569,A 0.000,B 0.000,C 90.000,E1 282.479} C_DIS
LIN {X -0.204,Y -459.230,Z 1237.565,A 0.000,B 0.000,C 90.000,E1 281.715} C_DIS
LIN {X -0.096,Y -461.219,Z 1237.562,A 0.000,B 0.000,C 90.000,E1 281.186} C_DIS
LIN {X 0.016,Y -462.943,Z 1237.559,A 0.000,B 0.000,C 90.000,E1 280.658} C_DIS
LIN {X 0.057,Y -464.412,Z 1237.556,A 0.000,B 0.000,C 90.000,E1 280.141} C_DIS
LIN {X 0.190,Y -465.650,Z 1237.554,A 0.000,B 0.000,C 90.000,E1 279.613} C_DIS
LIN {X -0.205,Y -466.587,Z 1237.551,A 0.000,B 0.000,C 90.000,E1 279.151} C_DIS
LIN {X -0.061,Y -467.246,Z 1237.548,A 0.000,B 0.000,C 90.000,E1 278.624} C_DIS
LIN {X 0.018,Y -467.571,Z 1237.545,A 0.000,B 0.000,C 90.000,E1 278.106} C_DIS
LIN {X 0.103,Y -467.600,Z 1237.542,A 0.000,B 0.000,C 90.000,E1 277.587} C_DIS
LIN {X 0.192,Y -467.205,Z 1237.539,A 0.000,B 0.000,C 90.000,E1 277.068} C_DIS
LIN {X -0.182,Y -466.370,Z 1237.537,A 0.000,B 0.000,C 90.000,E1 276.606} C_DIS
LIN {X -0.095,Y -465.095,Z 1237.534,A 0.000,B 0.000,C 90.000,E1 276.087} C_DIS
LIN {X -0.013,Y -463.442,Z 1237.531,A 0.000,B 0.000,C 90.000,E1 275.568} C_DIS
LIN {X -0.157,Y -460.114,Z 1237.527,A 0.000,B 0.000,C 90.000,E1 274.821} C_DIS
LIN {X -0.105,Y -457.252,Z 1237.524,A 0.000,B 0.000,C 90.000,E1 274.302} C_DIS
LIN {X 0.160,Y -455.612,Z 1237.522,A 0.000,B 0.000,C 90.000,E1 274.012} C_DIS
LIN {X 0.151,Y -451.596,Z 1237.520,A 0.000,B 0.000,C 90.000,E1 273.498} C_DIS
LIN {X 0.150,Y -446.575,Z 1237.517,A 0.000,B 0.000,C 90.000,E1 272.980} C_DIS
LIN {X -0.150,Y -440.414,Z 1237.514,A 0.000,B 0.000,C 90.000,E1 272.522} C_DIS
LIN {X 0.135,Y -433.845,Z 1237.512,A 0.000,B 0.000,C 90.000,E1 272.064} C_DIS
LIN {X 0.095,Y -426.926,Z 1237.510,A 0.000,B 0.000,C 90.000,E1 271.718} C_DIS
LIN {X 0.073,Y -419.872,Z 1237.508,A 0.000,B 0.000,C 90.000,E1 271.432} C_DIS
LIN {X 0.002,Y -412.971,Z 1237.507,A 0.000,B 0.000,C 90.000,E1 271.203} C_DIS
LIN {X 0.185,Y -405.850,Z 1237.506,A 0.000,B 0.000,C 90.000,E1 270.974} C_DIS
LIN {X 0.070,Y -394.855,Z 1237.504,A 0.000,B 0.000,C 90.000,E1 270.745} C_DIS
LIN {X -0.062,Y -387.123,Z 1237.503,A 0.000,B 0.000,C 90.000,E1 270.630} C_DIS
LIN {X -0.030,Y -378.027,Z 1237.503,A 0.000,B 0.000,C 90.000,E1 270.516} C_DIS
LIN {X -0.082,Y -366.693,Z 1237.502,A 0.000,B 0.000,C 90.000,E1 270.458} C_DIS
LIN {X -0.137,Y -362.262,Z 1237.502,A 0.000,B 0.000,C 90.000,E1 270.458} C_DIS
LIN {X 0.085,Y -181.573,Z 1237.502,A 0.000,B 0.000,C 90.000,E1 270.401} C_DIS
LIN {X -0.048,Y -180.905,Z 1237.474,A 0.000,B 0.000,C 90.000,E1 265.355} C_DIS
LIN {X 0.025,Y -180.674,Z 1237.469,A 0.000,B 0.000,C 90.000,E1 264.489} C_DIS
LIN {X -0.075,Y -178.756,Z 1237.441,A 0.000,B 0.000,C 90.000,E1 259.454} C_DIS
LIN {X -0.003,Y -175.803,Z 1237.413,A 0.000,B 0.000,C 90.000,E1 254.338} C_DIS
LIN {X -0.008,Y -171.988,Z 1237.385,A 0.000,B 0.000,C 90.000,E1 249.209} C_DIS
LIN {X 0.030,Y -171.398,Z 1237.380,A 0.000,B 0.000,C 90.000,E1 248.337} C_DIS
LIN {X 0.014,Y -167.640,Z 1237.356,A 0.000,B 0.000,C 90.000,E1 244.024} C_DIS
LIN {X 0.029,Y -166.300,Z 1237.346,A 0.000,B 0.000,C 90.000,E1 242.281} C_DIS
LIN {X 0.023,Y -163.044,Z 1237.327,A 0.000,B 0.000,C 90.000,E1 238.791} C_DIS
LIN {X -0.015,Y -160.976,Z 1237.312,A 0.000,B 0.000,C 90.000,E1 236.167} C_DIS
LIN {X -0.038,Y -157.727,Z 1237.292,A 0.000,B 0.000,C 90.000,E1 232.637} C_DIS
LIN {X -0.099,Y -155.766,Z 1237.277,A 0.000,B 0.000,C 90.000,E1 229.989} C_DIS
LIN {X -0.043,Y -152.022,Z 1237.253,A 0.000,B 0.000,C 90.000,E1 225.486} C_DIS
LIN {X -0.025,Y -150.270,Z 1237.238,A 0.000,B 0.000,C 90.000,E1 222.771} C_DIS
LIN {X -0.007,Y -147.021,Z 1237.212,A 0.000,B 0.000,C 90.000,E1 218.222} C_DIS
LIN {X 0.014,Y -145.604,Z 1237.197,A 0.000,B 0.000,C 90.000,E1 215.471} C_DIS
LIN {X 0.017,Y -142.989,Z 1237.172,A 0.000,B 0.000,C 90.000,E1 210.875} C_DIS
LIN {X 0.018,Y -141.617,Z 1237.151,A 0.000,B 0.000,C 90.000,E1 207.180} C_DIS
LIN {X 0.059,Y -139.429,Z 1237.115,A 0.000,B 0.000,C 90.000,E1 200.663} C_DIS
LIN {X -0.022,Y -139.159,Z 1237.105,A 0.000,B 0.000,C 90.000,E1 198.833} C_DIS
LIN {X -0.005,Y -138.342,Z 1237.058,A 0.000,B 0.000,C 90.000,E1 190.423} C_DIS
LIN {X -0.023,Y -139.480,Z 1237.006,A 0.000,B 0.000,C 90.000,E1 181.088} C_DIS
LIN {X 0.058,Y -141.069,Z 1236.975,A 0.000,B 0.000,C 90.000,E1 175.469} C_DIS
LIN {X 0.013,Y -142.444,Z 1236.959,A 0.000,B 0.000,C 90.000,E1 172.704} C_DIS
LIN {X -0.039,Y -144.684,Z 1236.934,A 0.000,B 0.000,C 90.000,E1 168.105} C_DIS
LIN {X 0.056,Y -147.274,Z 1236.913,A 0.000,B 0.000,C 90.000,E1 164.393} C_DIS
LIN {X -0.069,Y -150.592,Z 1236.888,A 0.000,B 0.000,C 90.000,E1 159.880} C_DIS
LIN {X 0.008,Y -154.065,Z 1236.868,A 0.000,B 0.000,C 90.000,E1 156.230} C_DIS
LIN {X 0.075,Y -157.484,Z 1236.848,A 0.000,B 0.000,C 90.000,E1 152.615} C_DIS
LIN {X 0.021,Y -161.709,Z 1236.828,A 0.000,B 0.000,C 90.000,E1 149.076} C_DIS
LIN {X 0.035,Y -165.903,Z 1236.809,A 0.000,B 0.000,C 90.000,E1 145.548} C_DIS
LIN {X 0.023,Y -170.888,Z 1236.789,A 0.000,B 0.000,C 90.000,E1 142.065} C_DIS
LIN {X 0.050,Y -175.756,Z 1236.770,A 0.000,B 0.000,C 90.000,E1 138.609} C_DIS
LIN {X -0.077,Y -181.365,Z 1236.751,A 0.000,B 0.000,C 90.000,E1 135.243} C_DIS
LIN {X 0.056,Y -186.859,Z 1236.733,A 0.000,B 0.000,C 90.000,E1 131.838} C_DIS
LIN {X 0.010,Y -191.444,Z 1236.719,A 0.000,B 0.000,C 90.000,E1 129.358} C_DIS
LIN {X -0.059,Y -197.297,Z 1236.700,A 0.000,B 0.000,C 90.000,E1 126.091} C_DIS
LIN {X 0.069,Y -200.764,Z 1236.691,A 0.000,B 0.000,C 90.000,E1 124.326} C_DIS
LIN {X 0.056,Y -309.965,Z 1236.691,A 0.000,B 0.000,C 90.000,E1 124.326} C_DIS
LIN {X -0.046,Y -311.749,Z 1236.691,A 0.000,B 0.000,C 90.000,E1 124.326} C_DIS
LIN {X 0.154,Y -316.099,Z 1236.690,A 0.000,B 0.000,C 90.000,E1 124.119} C_DIS
LIN {X -0.084,Y -318.432,Z 1236.689,A 0.000,B 0.000,C 90.000,E1 123.992} C_DIS
LIN {X 0.057,Y -321.608,Z 1236.687,A 0.000,B 0.000,C 90.000,E1 123.627} C_DIS
LIN {X -0.168,Y -323.579,Z 1236.685,A 0.000,B 0.000,C 90.000,E1 123.372} C_DIS
LIN {X 0.057,Y -325.121,Z 1236.684,A 0.000,B 0.000,C 90.000,E1 123.038} C_DIS
LIN {X -0.027,Y -327.561,Z 1236.680,A 0.000,B 0.000,C 90.000,E1 122.418} C_DIS
LIN {X 0.017,Y -338.377,Z 1236.664,A 0.000,B 0.000,C 90.000,E1 119.589} C_DIS
LIN {X 0.002,Y -350.570,Z 1236.649,A 0.000,B 0.000,C 90.000,E1 116.821} C_DIS
LIN {X 0.197,Y -364.239,Z 1236.634,A 0.000,B 0.000,C 90.000,E1 114.079} C_DIS
LIN {X -0.124,Y -377.728,Z 1236.621,A 0.000,B 0.000,C 90.000,E1 111.770} C_DIS
LIN {X -0.048,Y -392.577,Z 1236.608,A 0.000,B 0.000,C 90.000,E1 109.450} C_DIS
LIN {X -0.229,Y -408.886,Z 1236.595,A 0.000,B 0.000,C 90.000,E1 107.221} C_DIS
LIN {X -0.135,Y -426.773,Z 1236.583,A 0.000,B 0.000,C 90.000,E1 105.009} C_DIS
LIN {X -0.141,Y -446.239,Z 1236.571,A 0.000,B 0.000,C 90.000,E1 102.883} C_DIS
LIN {X 0.011,Y -466.474,Z 1236.561,A 0.000,B 0.000,C 90.000,E1 100.894} C_DIS
LIN {X 0.005,Y -474.044,Z 1236.557,A 0.000,B 0.000,C 90.000,E1 100.197} C_DIS
LIN {X -0.026,Y -475.951,Z 1236.555,A 0.000,B 0.000,C 90.000,E1 99.962} C_DIS
LIN {X -0.057,Y -477.400,Z 1236.554,A 0.000,B 0.000,C 90.000,E1 99.726} C_DIS
LIN {X 0.075,Y -479.374,Z 1236.551,A 0.000,B 0.000,C 90.000,E1 99.208} C_DIS
LIN {X -0.256,Y -480.219,Z 1236.548,A 0.000,B 0.000,C 90.000,E1 98.746} C_DIS
LIN {X -0.028,Y -480.082,Z 1236.546,A 0.000,B 0.000,C 90.000,E1 98.219} C_DIS
LIN {X 0.133,Y -478.945,Z 1236.543,A 0.000,B 0.000,C 90.000,E1 97.701} C_DIS
LIN {X 0.007,Y -477.949,Z 1236.542,A 0.000,B 0.000,C 90.000,E1 97.466} C_DIS
LIN {X -0.179,Y -476.604,Z 1236.540,A 0.000,B 0.000,C 90.000,E1 97.239} C_DIS
LIN {X 0.125,Y -456.613,Z 1236.525,A 0.000,B 0.000,C 90.000,E1 94.416} C_DIS
LIN {X -0.091,Y -435.940,Z 1236.507,A 0.000,B 0.000,C 90.000,E1 91.318} C_DIS
LIN {X -0.078,Y -421.889,Z 1236.494,A 0.000,B 0.000,C 90.000,E1 88.912} C_DIS
LIN {X 0.085,Y -407.506,Z 1236.479,A 0.000,B 0.000,C 90.000,E1 86.159} C_DIS
LIN {X 0.112,Y -398.834,Z 1236.469,A 0.000,B 0.000,C 90.000,E1 84.489} C_DIS
LIN {X -0.008,Y -388.654,Z 1236.458,A 0.000,B 0.000,C 90.000,E1 82.534} C_DIS
LIN {X 0.169,Y -379.803,Z 1236.449,A 0.000,B 0.000,C 90.000,E1 80.792} C_DIS
